LIN {X 0,Y 412.108,Z 841.021,A -85,B 0,C 180,E1 19370.746,E2 19370.746} C_VEL
LIN {X 0,Y 410.858,Z 854.484,A -85,B 0,C 180,E1 19368.885,E2 19368.885} C_VEL
LIN {X 0,Y 409.864,Z 866.557,A -85,B 0,C 180,E1 19366.876,E2 19366.876} C_VEL
LIN {X 0,Y 409.078,Z 878.045,A -85,B 0,C 180,E1 19364.559,E2 19364.559} C_VEL
LIN {X 0,Y 408.646,Z 887.648,A -85,B 0,C 180,E1 19362.147,E2 19362.147} C_VEL
LIN {X 0,Y 408.473,Z 895.28,A -85,B 0,C 180,E1 19359.724,E2 19359.724} C_VEL
LIN {X 0,Y 408.505,Z 901.076,A -85,B 0,C 180,E1 19357.312,E2 19357.312} C_VEL
LIN {X 0,Y 408.633,Z 905.166,A -85,B 0,C 180,E1 19354.913,E2 19354.913} C_VEL
LIN {X 0,Y 408.749,Z 907.618,A -85,B 0,C 180,E1 19352.524,E2 19352.524} C_VEL
LIN {X 0,Y 408.815,Z 908.485,A -85,B 0,C 180,E1 19350,E2 19350} C_VEL
LIN {X 0,Y 408.753,Z 907.591,A -85,B 0,C 180,E1 19347.477,E2 19347.477} C_VEL
LIN {X 0,Y 408.634,Z 904.94,A -85,B 0,C 180,E1 19344.947,E2 19344.947} C_VEL
LIN {X 0,Y 408.493,Z 900.479,A -85,B 0,C 180,E1 19342.405,E2 19342.405} C_VEL
LIN {X 0,Y 408.487,Z 894.1,A -85,B 0,C 180,E1 19339.85,E2 19339.85} C_VEL
LIN {X 0,Y 408.69,Z 886.166,A -85,B 0,C 180,E1 19337.424,E2 19337.424} C_VEL
LIN {X 0,Y 409.156,Z 876.808,A -85,B 0,C 180,E1 19335.132,E2 19335.132} C_VEL
LIN {X 0,Y 409.932,Z 866.006,A -85,B 0,C 180,E1 19332.964,E2 19332.964} C_VEL
LIN {X 0,Y 411.042,Z 853.158,A -85,B 0,C 180,E1 19330.829,E2 19330.829} C_VEL
LIN {X 0,Y 412.424,Z 839.094,A -85,B 0,C 180,E1 19328.899,E2 19328.899} C_VEL
LIN {X 0,Y 414.001,Z 823.32,A -85,B 0,C 180,E1 19327.118,E2 19327.118} C_VEL
LIN {X 0,Y 415.652,Z 807.137,A -85,B 0,C 180,E1 19325.635,E2 19325.635} C_VEL
LIN {X 0,Y 417.149,Z 790.974,A -85,B 0,C 180,E1 19324.441,E2 19324.441} C_VEL
LIN {X 0,Y 418.634,Z 773.451,A -85,B 0,C 180,E1 19323.428,E2 19323.428} C_VEL
LIN {X 0,Y 419.933,Z 754.838,A -85,B 0,C 180,E1 19322.636,E2 19322.636} C_VEL
LIN {X 0,Y 420.832,Z 735.86,A -85,B 0,C 180,E1 19322.104,E2 19322.104} C_VEL
LIN {X 0,Y 423.722,Z 562.823,A -85,B 0,C 180,E1 19319.088,E2 19319.088} C_VEL
LIN {X 0,Y 421.288,Z 541.067,A -85,B 0,C 180,E1 19318.453,E2 19318.453} C_VEL
LIN {X 0,Y 426.206,Z 498.135,A -85,B 0,C 180,E1 19314.092,E2 19314.092} C_VEL
LIN {X 0,Y 423.296,Z 488.09,A -85,B 0,C 180,E1 19312.623,E2 19312.623} C_VEL
LIN {X 0,Y 417.623,Z 472.168,A -85,B 0,C 180,E1 19310.008,E2 19310.008} C_VEL
LIN {X 0,Y 412.165,Z 458.735,A -85,B 0,C 180,E1 19307.516,E2 19307.516} C_VEL
LIN {X 0,Y 409.464,Z 451.977,A -85,B 0,C 180,E1 19306.115,E2 19306.115} C_VEL
LIN {X 0,Y 409.438,Z 451.787,A -85,B 0,C 180,E1 19302.187,E2 19302.187} C_VEL
LIN {X 0,Y 409.436,Z 451.789,A -85,B 0,C 180,E1 19298.336,E2 19298.336} C_VEL
LIN {X 0,Y 409.437,Z 451.796,A -85,B 0,C 180,E1 19294.34,E2 19294.34} C_VEL
LIN {X 0,Y 409.439,Z 451.796,A -85,B 0,C 180,E1 19290.364,E2 19290.364} C_VEL
LIN {X 0,Y 409.438,Z 451.794,A -85,B 0,C 180,E1 19286.544,E2 19286.544} C_VEL
LIN {X 0,Y 409.442,Z 451.791,A -85,B 0,C 180,E1 19282.544,E2 19282.544} C_VEL
LIN {X 0,Y 409.433,Z 451.782,A -85,B 0,C 180,E1 19278.646,E2 19278.646} C_VEL
LIN {X 0,Y 409.428,Z 451.775,A -85,B 0,C 180,E1 19274.713,E2 19274.713} C_VEL
LIN {X 0,Y 409.428,Z 451.787,A -85,B 0,C 180,E1 19270.838,E2 19270.838} C_VEL
LIN {X 0,Y 409.427,Z 451.797,A -85,B 0,C 180,E1 19266.872,E2 19266.872} C_VEL
LIN {X 0,Y 409.431,Z 451.793,A -85,B 0,C 180,E1 19262.939,E2 19262.939} C_VEL
LIN {X 0,Y 409.436,Z 451.78,A -85,B 0,C 180,E1 19259.02,E2 19259.02} C_VEL
LIN {X 0,Y 409.434,Z 451.779,A -85,B 0,C 180,E1 19255.097,E2 19255.097} C_VEL
LIN {X 0,Y 409.438,Z 451.784,A -85,B 0,C 180,E1 19251.291,E2 19251.291} C_VEL
LIN {X 0,Y 409.438,Z 451.789,A -85,B 0,C 180,E1 19247.303,E2 19247.303} C_VEL
LIN {X 0,Y 409.441,Z 451.792,A -85,B 0,C 180,E1 19243.398,E2 19243.398} C_VEL
LIN {X 0,Y 409.441,Z 451.788,A -85,B 0,C 180,E1 19239.411,E2 19239.411} C_VEL
LIN {X 0,Y 409.434,Z 451.786,A -85,B 0,C 180,E1 19235.625,E2 19235.625} C_VEL
LIN {X 0,Y 409.429,Z 451.795,A -85,B 0,C 180,E1 19231.721,E2 19231.721} C_VEL
LIN {X 0,Y 409.479,Z 452.064,A -85,B 0,C 180,E1 19229.358,E2 19229.358} C_VEL
LIN {X 0,Y 414.365,Z 466.013,A -85,B 0,C 180,E1 19226.106,E2 19226.106} C_VEL
LIN {X 0,Y 418.718,Z 480.117,A -85,B 0,C 180,E1 19223.125,E2 19223.125} C_VEL
LIN {X 0,Y 421.8,Z 492.439,A -85,B 0,C 180,E1 19220.734,E2 19220.734} C_VEL
LIN {X 0,Y 418.756,Z 520.346,A -85,B 0,C 180,E1 19216.54,E2 19216.54} C_VEL
LIN {X 0,Y 416.088,Z 548.549,A -85,B 0,C 180,E1 19212.379,E2 19212.379} C_VEL
LIN {X 0,Y 415.681,Z 554.248,A -85,B 0,C 180,E1 19211.576,E2 19211.576} C_VEL
LIN {X 0,Y 417.659,Z 564.451,A -85,B 0,C 180,E1 19211.173,E2 19211.173} C_VEL
LIN {X 0,Y 420.599,Z 581.405,A -85,B 0,C 180,E1 19210.622,E2 19210.622} C_VEL
LIN {X 0,Y 418.499,Z 678.205,A -85,B 0,C 180,E1 19208.79,E2 19208.79} C_VEL
LIN {X 0,Y 417.949,Z 694.436,A -85,B 0,C 180,E1 19208.216,E2 19208.216} C_VEL
LIN {X 0,Y 417.211,Z 708.122,A -85,B 0,C 180,E1 19207.497,E2 19207.497} C_VEL
LIN {X 0,Y 416.181,Z 722.203,A -85,B 0,C 180,E1 19206.492,E2 19206.492} C_VEL
LIN {X 0,Y 415.036,Z 734.8,A -85,B 0,C 180,E1 19205.322,E2 19205.322} C_VEL
LIN {X 0,Y 413.801,Z 747.225,A -85,B 0,C 180,E1 19203.845,E2 19203.845} C_VEL
LIN {X 0,Y 412.619,Z 757.902,A -85,B 0,C 180,E1 19202.215,E2 19202.215} C_VEL
LIN {X 0,Y 411.608,Z 766.741,A -85,B 0,C 180,E1 19200.51,E2 19200.51} C_VEL
LIN {X 0,Y 410.668,Z 774.752,A -85,B 0,C 180,E1 19198.485,E2 19198.485} C_VEL
LIN {X 0,Y 409.991,Z 780.564,A -85,B 0,C 180,E1 19196.489,E2 19196.489} C_VEL
LIN {X 0,Y 409.526,Z 784.81,A -85,B 0,C 180,E1 19194.369,E2 19194.369} C_VEL
LIN {X 0,Y 409.251,Z 787.256,A -85,B 0,C 180,E1 19192.187,E2 19192.187} C_VEL
LIN {X 0,Y 409.145,Z 787.957,A -85,B 0,C 180,E1 19190.006,E2 19190.006} C_VEL
LIN {X 0,Y 409.137,Z 787.808,A -85,B 0,C 180,E1 19189.341,E2 19189.341} C_VEL
LIN {X 0,Y 408.18,Z 787.446,A -85,B 0,C 180,E1 19188.262,E2 19188.262} C_VEL
LIN {X 0,Y 404.232,Z 786.122,A -85,B 0,C 180,E1 19186.459,E2 19186.459} C_VEL
LIN {X 0,Y 401.873,Z 784.219,A -85,B 0,C 180,E1 19185.094,E2 19185.094} C_VEL
LIN {X 0,Y 401.627,Z 783.02,A -85,B 0,C 180,E1 19184.483,E2 19184.483} C_VEL
LIN {X 0,Y 402.092,Z 777.918,A -85,B 0,C 180,E1 19182.494,E2 19182.494} C_VEL
LIN {X 0,Y 402.798,Z 770.631,A -85,B 0,C 180,E1 19180.44,E2 19180.44} C_VEL
LIN {X 0,Y 403.609,Z 762.582,A -85,B 0,C 180,E1 19178.691,E2 19178.691} C_VEL
LIN {X 0,Y 404.628,Z 752.359,A -85,B 0,C 180,E1 19176.954,E2 19176.954} C_VEL
LIN {X 0,Y 405.691,Z 741.112,A -85,B 0,C 180,E1 19175.444,E2 19175.444} C_VEL
LIN {X 0,Y 406.794,Z 728.273,A -85,B 0,C 180,E1 19174.087,E2 19174.087} C_VEL
LIN {X 0,Y 407.821,Z 714.219,A -85,B 0,C 180,E1 19172.951,E2 19172.951} C_VEL
LIN {X 0,Y 408.63,Z 700.315,A -85,B 0,C 180,E1 19172.103,E2 19172.103} C_VEL
LIN {X 0,Y 409.274,Z 683.774,A -85,B 0,C 180,E1 19171.408,E2 19171.408} C_VEL
LIN {X 0,Y 409.627,Z 665.81,A -85,B 0,C 180,E1 19170.979,E2 19170.979} C_VEL
LIN {X 0,Y 411.05,Z 579.361,A -85,B 0,C 180,E1 19169.384,E2 19169.384} C_VEL
LIN {X 0,Y 406.705,Z 554.518,A -85,B 0,C 180,E1 19168.626,E2 19168.626} C_VEL
LIN {X 0,Y 408.776,Z 527.92,A -85,B 0,C 180,E1 19164.807,E2 19164.807} C_VEL
LIN {X 0,Y 411.265,Z 500.481,A -85,B 0,C 180,E1 19160.766,E2 19160.766} C_VEL
LIN {X 0,Y 412.101,Z 490.248,A -85,B 0,C 180,E1 19159.232,E2 19159.232} C_VEL
LIN {X 0,Y 407.297,Z 472.284,A -85,B 0,C 180,E1 19155.934,E2 19155.934} C_VEL
LIN {X 0,Y 402.224,Z 455.434,A -85,B 0,C 180,E1 19152.644,E2 19152.644} C_VEL
LIN {X 0,Y 401.461,Z 452.888,A -85,B 0,C 180,E1 19152.063,E2 19152.063} C_VEL
LIN {X 0,Y 401.432,Z 452.768,A -85,B 0,C 180,E1 19148.215,E2 19148.215} C_VEL
LIN {X 0,Y 401.43,Z 452.789,A -85,B 0,C 180,E1 19144.317,E2 19144.317} C_VEL
LIN {X 0,Y 401.426,Z 452.793,A -85,B 0,C 180,E1 19140.376,E2 19140.376} C_VEL
LIN {X 0,Y 401.426,Z 452.791,A -85,B 0,C 180,E1 19136.43,E2 19136.43} C_VEL
LIN {X 0,Y 401.437,Z 452.779,A -85,B 0,C 180,E1 19132.574,E2 19132.574} C_VEL
LIN {X 0,Y 401.467,Z 452.776,A -85,B 0,C 180,E1 19128.89,E2 19128.89} C_VEL
LIN {X 0,Y 401.477,Z 452.791,A -85,B 0,C 180,E1 19124.985,E2 19124.985} C_VEL
LIN {X 0,Y 401.488,Z 452.764,A -85,B 0,C 180,E1 19120.918,E2 19120.918} C_VEL
LIN {X 0,Y 401.487,Z 452.782,A -85,B 0,C 180,E1 19116.925,E2 19116.925} C_VEL
LIN {X 0,Y 401.485,Z 452.766,A -85,B 0,C 180,E1 19112.882,E2 19112.882} C_VEL
LIN {X 0,Y 401.478,Z 452.783,A -85,B 0,C 180,E1 19109.055,E2 19109.055} C_VEL
LIN {X 0,Y 401.461,Z 452.761,A -85,B 0,C 180,E1 19105.207,E2 19105.207} C_VEL
LIN {X 0,Y 401.452,Z 452.789,A -85,B 0,C 180,E1 19101.477,E2 19101.477} C_VEL
LIN {X 0,Y 401.449,Z 452.752,A -85,B 0,C 180,E1 19097.54,E2 19097.54} C_VEL
LIN {X 0,Y 401.456,Z 452.787,A -85,B 0,C 180,E1 19093.54,E2 19093.54} C_VEL
LIN {X 0,Y 401.458,Z 452.761,A -85,B 0,C 180,E1 19089.606,E2 19089.606} C_VEL
LIN {X 0,Y 401.469,Z 452.782,A -85,B 0,C 180,E1 19085.718,E2 19085.718} C_VEL
LIN {X 0,Y 401.48,Z 452.768,A -85,B 0,C 180,E1 19081.856,E2 19081.856} C_VEL
LIN {X 0,Y 401.496,Z 452.774,A -85,B 0,C 180,E1 19078.002,E2 19078.002} C_VEL
LIN {X 0,Y 401.502,Z 452.771,A -85,B 0,C 180,E1 19073.997,E2 19073.997} C_VEL
LIN {X 0,Y 401.502,Z 452.774,A -85,B 0,C 180,E1 19070.106,E2 19070.106} C_VEL
LIN {X 0,Y 401.502,Z 452.768,A -85,B 0,C 180,E1 19066.169,E2 19066.169} C_VEL
LIN {X 0,Y 401.5,Z 452.785,A -85,B 0,C 180,E1 19062.163,E2 19062.163} C_VEL
LIN {X 0,Y 401.497,Z 452.766,A -85,B 0,C 180,E1 19058.219,E2 19058.219} C_VEL
LIN {X 0,Y 401.488,Z 452.779,A -85,B 0,C 180,E1 19054.321,E2 19054.321} C_VEL
LIN {X 0,Y 401.488,Z 452.789,A -85,B 0,C 180,E1 19050.36,E2 19050.36} C_VEL
LIN {X 0,Y 401.485,Z 452.785,A -85,B 0,C 180,E1 19046.436,E2 19046.436} C_VEL
LIN {X 0,Y 401.484,Z 452.786,A -85,B 0,C 180,E1 19042.58,E2 19042.58} C_VEL
LIN {X 0,Y 401.489,Z 452.787,A -85,B 0,C 180,E1 19038.556,E2 19038.556} C_VEL
LIN {X 0,Y 401.49,Z 452.779,A -85,B 0,C 180,E1 19034.582,E2 19034.582} C_VEL
LIN {X 0,Y 401.526,Z 453.016,A -85,B 0,C 180,E1 19032.727,E2 19032.727} C_VEL
LIN {X 0,Y 408.421,Z 472.022,A -85,B 0,C 180,E1 19029.664,E2 19029.664} C_VEL
LIN {X 0,Y 415.923,Z 494.073,A -85,B 0,C 180,E1 19026.463,E2 19026.463} C_VEL
LIN {X 0,Y 417.225,Z 498.2,A -85,B 0,C 180,E1 19025.904,E2 19025.904} C_VEL
LIN {X 0,Y 412.81,Z 540.992,A -85,B 0,C 180,E1 19021.622,E2 19021.622} C_VEL
LIN {X 0,Y 415.431,Z 566.716,A -85,B 0,C 180,E1 19020.959,E2 19020.959} C_VEL
LIN {X 0,Y 412.493,Z 738.8,A -85,B 0,C 180,E1 19017.967,E2 19017.967} C_VEL
LIN {X 0,Y 411.552,Z 757.391,A -85,B 0,C 180,E1 19017.403,E2 19017.403} C_VEL
LIN {X 0,Y 410.372,Z 774.696,A -85,B 0,C 180,E1 19016.636,E2 19016.636} C_VEL
LIN {X 0,Y 408.983,Z 791.545,A -85,B 0,C 180,E1 19015.641,E2 19015.641} C_VEL
LIN {X 0,Y 407.427,Z 808.616,A -85,B 0,C 180,E1 19014.349,E2 19014.349} C_VEL
LIN {X 0,Y 405.858,Z 824.312,A -85,B 0,C 180,E1 19012.872,E2 19012.872} C_VEL
LIN {X 0,Y 404.35,Z 839.602,A -85,B 0,C 180,E1 19011.11,E2 19011.11} C_VEL
LIN {X 0,Y 403.013,Z 853.315,A -85,B 0,C 180,E1 19009.192,E2 19009.192} C_VEL
LIN {X 0,Y 401.932,Z 865.851,A -85,B 0,C 180,E1 19007.07,E2 19007.07} C_VEL
LIN {X 0,Y 401.161,Z 876.529,A -85,B 0,C 180,E1 19004.876,E2 19004.876} C_VEL
LIN {X 0,Y 400.687,Z 886.318,A -85,B 0,C 180,E1 19002.392,E2 19002.392} C_VEL
LIN {X 0,Y 400.51,Z 894.001,A -85,B 0,C 180,E1 18999.919,E2 18999.919} C_VEL
LIN {X 0,Y 400.548,Z 899.837,A -85,B 0,C 180,E1 18997.459,E2 18997.459} C_VEL
LIN {X 0,Y 400.697,Z 903.962,A -85,B 0,C 180,E1 18995.011,E2 18995.011} C_VEL
LIN {X 0,Y 400.836,Z 906.525,A -85,B 0,C 180,E1 18992.431,E2 18992.431} C_VEL
LIN {X 0,Y 400.897,Z 907.312,A -85,B 0,C 180,E1 18989.857,E2 18989.857} C_VEL
LIN {X 0,Y 400.823,Z 906.329,A -85,B 0,C 180,E1 18987.284,E2 18987.284} C_VEL
LIN {X 0,Y 400.676,Z 903.574,A -85,B 0,C 180,E1 18984.703,E2 18984.703} C_VEL
LIN {X 0,Y 400.524,Z 898.987,A -85,B 0,C 180,E1 18982.109,E2 18982.109} C_VEL
LIN {X 0,Y 400.516,Z 892.781,A -85,B 0,C 180,E1 18979.606,E2 18979.606} C_VEL
LIN {X 0,Y 400.732,Z 884.94,A -85,B 0,C 180,E1 18977.17,E2 18977.17} C_VEL
LIN {X 0,Y 401.238,Z 875.583,A -85,B 0,C 180,E1 18974.832,E2 18974.832} C_VEL
LIN {X 0,Y 402.063,Z 864.886,A -85,B 0,C 180,E1 18972.638,E2 18972.638} C_VEL
LIN {X 0,Y 403.172,Z 852.878,A -85,B 0,C 180,E1 18970.591,E2 18970.591} C_VEL
LIN {X 0,Y 404.624,Z 838.96,A -85,B 0,C 180,E1 18968.624,E2 18968.624} C_VEL
LIN {X 0,Y 406.209,Z 824.047,A -85,B 0,C 180,E1 18966.884,E2 18966.884} C_VEL
LIN {X 0,Y 408.013,Z 807.384,A -85,B 0,C 180,E1 18965.303,E2 18965.303} C_VEL
LIN {X 0,Y 409.667,Z 790.598,A -85,B 0,C 180,E1 18964.028,E2 18964.028} C_VEL
LIN {X 0,Y 411.178,Z 773.845,A -85,B 0,C 180,E1 18963.031,E2 18963.031} C_VEL
LIN {X 0,Y 412.528,Z 755.816,A -85,B 0,C 180,E1 18962.229,E2 18962.229} C_VEL
LIN {X 0,Y 413.534,Z 737.11,A -85,B 0,C 180,E1 18961.667,E2 18961.667} C_VEL
LIN {X 0,Y 416.67,Z 563.768,A -85,B 0,C 180,E1 18958.584,E2 18958.584} C_VEL
LIN {X 0,Y 414.152,Z 541.339,A -85,B 0,C 180,E1 18957.918,E2 18957.918} C_VEL
LIN {X 0,Y 419.123,Z 500.336,A -85,B 0,C 180,E1 18953.662,E2 18953.662} C_VEL
LIN {X 0,Y 413.776,Z 483.941,A -85,B 0,C 180,E1 18951.078,E2 18951.078} C_VEL
LIN {X 0,Y 407.629,Z 467.636,A -85,B 0,C 180,E1 18948.151,E2 18948.151} C_VEL
LIN {X 0,Y 402.535,Z 455.853,A -85,B 0,C 180,E1 18945.735,E2 18945.735} C_VEL
LIN {X 0,Y 401.519,Z 452.934,A -85,B 0,C 180,E1 18945.053,E2 18945.053} C_VEL
LIN {X 0,Y 401.506,Z 452.783,A -85,B 0,C 180,E1 18941.014,E2 18941.014} C_VEL
LIN {X 0,Y 401.496,Z 452.785,A -85,B 0,C 180,E1 18937.06,E2 18937.06} C_VEL
LIN {X 0,Y 401.494,Z 452.777,A -85,B 0,C 180,E1 18933.051,E2 18933.051} C_VEL
LIN {X 0,Y 401.493,Z 452.775,A -85,B 0,C 180,E1 18929.053,E2 18929.053} C_VEL
LIN {X 0,Y 401.491,Z 452.778,A -85,B 0,C 180,E1 18925.047,E2 18925.047} C_VEL
LIN {X 0,Y 401.491,Z 452.782,A -85,B 0,C 180,E1 18921.015,E2 18921.015} C_VEL
LIN {X 0,Y 401.49,Z 452.787,A -85,B 0,C 180,E1 18917.001,E2 18917.001} C_VEL
LIN {X 0,Y 401.492,Z 452.777,A -85,B 0,C 180,E1 18913.098,E2 18913.098} C_VEL
LIN {X 0,Y 401.493,Z 452.767,A -85,B 0,C 180,E1 18909.171,E2 18909.171} C_VEL
LIN {X 0,Y 401.496,Z 452.767,A -85,B 0,C 180,E1 18905.287,E2 18905.287} C_VEL
LIN {X 0,Y 401.502,Z 452.779,A -85,B 0,C 180,E1 18901.284,E2 18901.284} C_VEL
LIN {X 0,Y 401.499,Z 452.787,A -85,B 0,C 180,E1 18897.288,E2 18897.288} C_VEL
LIN {X 0,Y 401.503,Z 452.78,A -85,B 0,C 180,E1 18893.278,E2 18893.278} C_VEL
LIN {X 0,Y 401.499,Z 452.776,A -85,B 0,C 180,E1 18889.235,E2 18889.235} C_VEL
LIN {X 0,Y 401.502,Z 452.774,A -85,B 0,C 180,E1 18885.285,E2 18885.285} C_VEL
LIN {X 0,Y 401.501,Z 452.778,A -85,B 0,C 180,E1 18881.261,E2 18881.261} C_VEL
LIN {X 0,Y 401.506,Z 452.785,A -85,B 0,C 180,E1 18877.294,E2 18877.294} C_VEL
LIN {X 0,Y 401.5,Z 452.78,A -85,B 0,C 180,E1 18873.368,E2 18873.368} C_VEL
LIN {X 0,Y 401.536,Z 453.052,A -85,B 0,C 180,E1 18870.359,E2 18870.359} C_VEL
LIN {X 0,Y 406.172,Z 465.882,A -85,B 0,C 180,E1 18867.209,E2 18867.209} C_VEL
LIN {X 0,Y 410.698,Z 480.056,A -85,B 0,C 180,E1 18864.075,E2 18864.075} C_VEL
LIN {X 0,Y 414.48,Z 494.529,A -85,B 0,C 180,E1 18861.155,E2 18861.155} C_VEL
LIN {X 0,Y 412.074,Z 516.12,A -85,B 0,C 180,E1 18857.839,E2 18857.839} C_VEL
LIN {X 0,Y 409.252,Z 543.685,A -85,B 0,C 180,E1 18853.683,E2 18853.683} C_VEL
LIN {X 0,Y 408.353,Z 554.376,A -85,B 0,C 180,E1 18852.136,E2 18852.136} C_VEL
LIN {X 0,Y 413.566,Z 581.773,A -85,B 0,C 180,E1 18851.143,E2 18851.143} C_VEL
LIN {X 0,Y 411.336,Z 678.782,A -85,B 0,C 180,E1 18849.276,E2 18849.276} C_VEL
LIN {X 0,Y 410.757,Z 694.919,A -85,B 0,C 180,E1 18848.698,E2 18848.698} C_VEL
LIN {X 0,Y 409.931,Z 709.332,A -85,B 0,C 180,E1 18847.926,E2 18847.926} C_VEL
LIN {X 0,Y 408.832,Z 723.463,A -85,B 0,C 180,E1 18846.895,E2 18846.895} C_VEL
LIN {X 0,Y 407.627,Z 735.875,A -85,B 0,C 180,E1 18845.717,E2 18845.717} C_VEL
LIN {X 0,Y 406.313,Z 748.189,A -85,B 0,C 180,E1 18844.224,E2 18844.224} C_VEL
LIN {X 0,Y 405.035,Z 758.912,A -85,B 0,C 180,E1 18842.557,E2 18842.557} C_VEL
LIN {X 0,Y 403.933,Z 767.836,A -85,B 0,C 180,E1 18840.802,E2 18840.802} C_VEL
LIN {X 0,Y 402.929,Z 775.709,A -85,B 0,C 180,E1 18838.777,E2 18838.777} C_VEL
LIN {X 0,Y 402.189,Z 781.578,A -85,B 0,C 180,E1 18836.742,E2 18836.742} C_VEL
LIN {X 0,Y 401.667,Z 785.892,A -85,B 0,C 180,E1 18834.564,E2 18834.564} C_VEL
LIN {X 0,Y 401.366,Z 788.34,A -85,B 0,C 180,E1 18832.404,E2 18832.404} C_VEL
LIN {X 0,Y 401.234,Z 789.138,A -85,B 0,C 180,E1 18830.114,E2 18830.114} C_VEL
LIN {X 0,Y 401.257,Z 788.058,A -85,B 0,C 180,E1 18827.846,E2 18827.846} C_VEL
LIN {X 0,Y 401.44,Z 785.457,A -85,B 0,C 180,E1 18825.752,E2 18825.752} C_VEL
LIN {X 0,Y 401.627,Z 783.02,A -85,B 0,C 180,E1 18824.483,E2 18824.483} C_VEL
LIN {X 0,Y 400.869,Z 780.731,A -85,B 0,C 180,E1 18823.427,E2 18823.427} C_VEL
LIN {X 0,Y 397.327,Z 776.403,A -85,B 0,C 180,E1 18821.672,E2 18821.672} C_VEL
LIN {X 0,Y 395.285,Z 772.231,A -85,B 0,C 180,E1 18820.385,E2 18820.385} C_VEL
LIN {X 0,Y 395.166,Z 769.988,A -85,B 0,C 180,E1 18819.829,E2 18819.829} C_VEL
LIN {X 0,Y 396.107,Z 761.081,A -85,B 0,C 180,E1 18817.98,E2 18817.98} C_VEL
LIN {X 0,Y 397.189,Z 750.691,A -85,B 0,C 180,E1 18816.286,E2 18816.286} C_VEL
LIN {X 0,Y 398.347,Z 738.786,A -85,B 0,C 180,E1 18814.751,E2 18814.751} C_VEL
LIN {X 0,Y 399.478,Z 725.741,A -85,B 0,C 180,E1 18813.444,E2 18813.444} C_VEL
LIN {X 0,Y 400.504,Z 711.738,A -85,B 0,C 180,E1 18812.361,E2 18812.361} C_VEL
LIN {X 0,Y 401.349,Z 696.534,A -85,B 0,C 180,E1 18811.499,E2 18811.499} C_VEL
LIN {X 0,Y 401.896,Z 681.019,A -85,B 0,C 180,E1 18810.909,E2 18810.909} C_VEL
LIN {X 0,Y 402.432,Z 653.413,A -85,B 0,C 180,E1 18810.324,E2 18810.324} C_VEL
LIN {X 0,Y 403.659,Z 580.369,A -85,B 0,C 180,E1 18808.957,E2 18808.957} C_VEL
LIN {X 0,Y 399.141,Z 554.231,A -85,B 0,C 180,E1 18808.134,E2 18808.134} C_VEL
LIN {X 0,Y 401.425,Z 526.958,A -85,B 0,C 180,E1 18804.138,E2 18804.138} C_VEL
LIN {X 0,Y 404.097,Z 499.455,A -85,B 0,C 180,E1 18800.026,E2 18800.026} C_VEL
LIN {X 0,Y 404.665,Z 492.91,A -85,B 0,C 180,E1 18799.032,E2 18799.032} C_VEL
LIN {X 0,Y 400.117,Z 475.734,A -85,B 0,C 180,E1 18795.824,E2 18795.824} C_VEL
LIN {X 0,Y 395.046,Z 458.853,A -85,B 0,C 180,E1 18792.471,E2 18792.471} C_VEL
LIN {X 0,Y 393.548,Z 453.877,A -85,B 0,C 180,E1 18791.381,E2 18791.381} C_VEL
LIN {X 0,Y 393.544,Z 453.735,A -85,B 0,C 180,E1 18787.44,E2 18787.44} C_VEL
LIN {X 0,Y 393.536,Z 453.78,A -85,B 0,C 180,E1 18783.423,E2 18783.423} C_VEL
LIN {X 0,Y 393.533,Z 453.779,A -85,B 0,C 180,E1 18779.459,E2 18779.459} C_VEL
LIN {X 0,Y 393.527,Z 453.781,A -85,B 0,C 180,E1 18775.408,E2 18775.408} C_VEL
LIN {X 0,Y 393.535,Z 453.774,A -85,B 0,C 180,E1 18771.316,E2 18771.316} C_VEL
LIN {X 0,Y 393.516,Z 453.758,A -85,B 0,C 180,E1 18767.464,E2 18767.464} C_VEL
LIN {X 0,Y 393.508,Z 453.779,A -85,B 0,C 180,E1 18763.601,E2 18763.601} C_VEL
LIN {X 0,Y 393.501,Z 453.77,A -85,B 0,C 180,E1 18759.816,E2 18759.816} C_VEL
LIN {X 0,Y 393.501,Z 453.769,A -85,B 0,C 180,E1 18755.849,E2 18755.849} C_VEL
LIN {X 0,Y 393.506,Z 453.773,A -85,B 0,C 180,E1 18751.905,E2 18751.905} C_VEL
LIN {X 0,Y 393.512,Z 453.765,A -85,B 0,C 180,E1 18748.039,E2 18748.039} C_VEL
LIN {X 0,Y 393.522,Z 453.767,A -85,B 0,C 180,E1 18744.147,E2 18744.147} C_VEL
LIN {X 0,Y 393.546,Z 453.766,A -85,B 0,C 180,E1 18740.364,E2 18740.364} C_VEL
LIN {X 0,Y 393.551,Z 453.746,A -85,B 0,C 180,E1 18736.38,E2 18736.38} C_VEL
LIN {X 0,Y 393.558,Z 453.772,A -85,B 0,C 180,E1 18732.471,E2 18732.471} C_VEL
LIN {X 0,Y 393.557,Z 453.738,A -85,B 0,C 180,E1 18728.474,E2 18728.474} C_VEL
LIN {X 0,Y 393.555,Z 453.776,A -85,B 0,C 180,E1 18724.517,E2 18724.517} C_VEL
LIN {X 0,Y 393.559,Z 453.74,A -85,B 0,C 180,E1 18720.437,E2 18720.437} C_VEL
LIN {X 0,Y 393.55,Z 453.775,A -85,B 0,C 180,E1 18716.505,E2 18716.505} C_VEL
LIN {X 0,Y 393.543,Z 453.748,A -85,B 0,C 180,E1 18712.555,E2 18712.555} C_VEL
LIN {X 0,Y 393.543,Z 453.776,A -85,B 0,C 180,E1 18708.57,E2 18708.57} C_VEL
LIN {X 0,Y 393.536,Z 453.751,A -85,B 0,C 180,E1 18704.679,E2 18704.679} C_VEL
LIN {X 0,Y 393.54,Z 453.777,A -85,B 0,C 180,E1 18700.714,E2 18700.714} C_VEL
LIN {X 0,Y 393.539,Z 453.769,A -85,B 0,C 180,E1 18696.809,E2 18696.809} C_VEL
LIN {X 0,Y 393.538,Z 453.757,A -85,B 0,C 180,E1 18692.779,E2 18692.779} C_VEL
LIN {X 0,Y 393.544,Z 453.764,A -85,B 0,C 180,E1 18688.782,E2 18688.782} C_VEL
LIN {X 0,Y 393.545,Z 453.767,A -85,B 0,C 180,E1 18684.78,E2 18684.78} C_VEL
LIN {X 0,Y 393.548,Z 453.765,A -85,B 0,C 180,E1 18680.757,E2 18680.757} C_VEL
LIN {X 0,Y 393.555,Z 453.769,A -85,B 0,C 180,E1 18676.815,E2 18676.815} C_VEL
LIN {X 0,Y 393.597,Z 454.026,A -85,B 0,C 180,E1 18673.457,E2 18673.457} C_VEL
LIN {X 0,Y 400.542,Z 473.077,A -85,B 0,C 180,E1 18670.281,E2 18670.281} C_VEL
LIN {X 0,Y 407.843,Z 494.443,A -85,B 0,C 180,E1 18667.092,E2 18667.092} C_VEL
LIN {X 0,Y 409.804,Z 500.937,A -85,B 0,C 180,E1 18666.189,E2 18666.189} C_VEL
LIN {X 0,Y 405.429,Z 541.304,A -85,B 0,C 180,E1 18662.077,E2 18662.077} C_VEL
LIN {X 0,Y 408.091,Z 567.582,A -85,B 0,C 180,E1 18661.393,E2 18661.393} C_VEL
LIN {X 0,Y 405.048,Z 738.109,A -85,B 0,C 180,E1 18658.387,E2 18658.387} C_VEL
LIN {X 0,Y 404.074,Z 756.704,A -85,B 0,C 180,E1 18657.813,E2 18657.813} C_VEL
LIN {X 0,Y 402.817,Z 774.328,A -85,B 0,C 180,E1 18657.016,E2 18657.016} C_VEL
LIN {X 0,Y 401.261,Z 792.231,A -85,B 0,C 180,E1 18655.925,E2 18655.925} C_VEL
LIN {X 0,Y 399.659,Z 808.92,A -85,B 0,C 180,E1 18654.617,E2 18654.617} C_VEL
LIN {X 0,Y 397.995,Z 824.776,A -85,B 0,C 180,E1 18653.074,E2 18653.074} C_VEL
LIN {X 0,Y 396.453,Z 839.691,A -85,B 0,C 180,E1 18651.295,E2 18651.295} C_VEL
LIN {X 0,Y 395.087,Z 853.081,A -85,B 0,C 180,E1 18649.362,E2 18649.362} C_VEL
LIN {X 0,Y 393.94,Z 865.854,A -85,B 0,C 180,E1 18647.123,E2 18647.123} C_VEL
LIN {X 0,Y 393.162,Z 876.344,A -85,B 0,C 180,E1 18644.884,E2 18644.884} C_VEL
LIN {X 0,Y 392.713,Z 885.455,A -85,B 0,C 180,E1 18642.499,E2 18642.499} C_VEL
LIN {X 0,Y 392.544,Z 893.096,A -85,B 0,C 180,E1 18639.974,E2 18639.974} C_VEL
LIN {X 0,Y 392.598,Z 898.872,A -85,B 0,C 180,E1 18637.463,E2 18637.463} C_VEL
LIN {X 0,Y 392.77,Z 902.929,A -85,B 0,C 180,E1 18634.966,E2 18634.966} C_VEL
LIN {X 0,Y 392.914,Z 905.343,A -85,B 0,C 180,E1 18632.48,E2 18632.48} C_VEL
LIN {X 0,Y 392.988,Z 906.14,A -85,B 0,C 180,E1 18630,E2 18630} C_VEL
LIN {X 0,Y 392.915,Z 905.337,A -85,B 0,C 180,E1 18627.521,E2 18627.521} C_VEL
LIN {X 0,Y 392.768,Z 902.957,A -85,B 0,C 180,E1 18625.035,E2 18625.035} C_VEL
LIN {X 0,Y 392.589,Z 898.957,A -85,B 0,C 180,E1 18622.537,E2 18622.537} C_VEL
LIN {X 0,Y 392.528,Z 893.275,A -85,B 0,C 180,E1 18620.026,E2 18620.026} C_VEL
LIN {X 0,Y 392.695,Z 885.785,A -85,B 0,C 180,E1 18617.501,E2 18617.501} C_VEL
LIN {X 0,Y 393.191,Z 876.288,A -85,B 0,C 180,E1 18614.967,E2 18614.967} C_VEL
LIN {X 0,Y 394.092,Z 865.066,A -85,B 0,C 180,E1 18612.546,E2 18612.546} C_VEL
LIN {X 0,Y 395.311,Z 852.598,A -85,B 0,C 180,E1 18610.343,E2 18610.343} C_VEL
LIN {X 0,Y 396.834,Z 838.825,A -85,B 0,C 180,E1 18608.339,E2 18608.339} C_VEL
LIN {X 0,Y 398.501,Z 824.099,A -85,B 0,C 180,E1 18606.567,E2 18606.567} C_VEL
LIN {X 0,Y 400.302,Z 808.551,A -85,B 0,C 180,E1 18605.032,E2 18605.032} C_VEL
LIN {X 0,Y 402.038,Z 792.182,A -85,B 0,C 180,E1 18603.725,E2 18603.725} C_VEL
LIN {X 0,Y 403.705,Z 774.988,A -85,B 0,C 180,E1 18602.65,E2 18602.65} C_VEL
LIN {X 0,Y 405.199,Z 756.378,A -85,B 0,C 180,E1 18601.786,E2 18601.786} C_VEL
LIN {X 0,Y 406.276,Z 737.933,A -85,B 0,C 180,E1 18601.206,E2 18601.206} C_VEL
LIN {X 0,Y 407.13,Z 697.172,A -85,B 0,C 180,E1 18600.456,E2 18600.456} C_VEL
LIN {X 0,Y 409.654,Z 564.686,A -85,B 0,C 180,E1 18598.06,E2 18598.06} C_VEL
LIN {X 0,Y 407.071,Z 541.874,A -85,B 0,C 180,E1 18597.375,E2 18597.375} C_VEL
LIN {X 0,Y 412.013,Z 503.231,A -85,B 0,C 180,E1 18593.296,E2 18593.296} C_VEL
LIN {X 0,Y 406.716,Z 486.818,A -85,B 0,C 180,E1 18590.635,E2 18590.635} C_VEL
LIN {X 0,Y 400.899,Z 471.491,A -85,B 0,C 180,E1 18587.793,E2 18587.793} C_VEL
LIN {X 0,Y 396.029,Z 460.11,A -85,B 0,C 180,E1 18585.395,E2 18585.395} C_VEL
LIN {X 0,Y 393.583,Z 453.942,A -85,B 0,C 180,E1 18583.966,E2 18583.966} C_VEL
LIN {X 0,Y 393.563,Z 453.767,A -85,B 0,C 180,E1 18579.997,E2 18579.997} C_VEL
LIN {X 0,Y 393.557,Z 453.761,A -85,B 0,C 180,E1 18575.935,E2 18575.935} C_VEL
LIN {X 0,Y 393.56,Z 453.759,A -85,B 0,C 180,E1 18571.947,E2 18571.947} C_VEL
LIN {X 0,Y 393.561,Z 453.756,A -85,B 0,C 180,E1 18568.034,E2 18568.034} C_VEL
LIN {X 0,Y 393.56,Z 453.755,A -85,B 0,C 180,E1 18563.984,E2 18563.984} C_VEL
LIN {X 0,Y 393.56,Z 453.757,A -85,B 0,C 180,E1 18559.949,E2 18559.949} C_VEL
LIN {X 0,Y 393.562,Z 453.765,A -85,B 0,C 180,E1 18555.925,E2 18555.925} C_VEL
LIN {X 0,Y 393.561,Z 453.775,A -85,B 0,C 180,E1 18551.875,E2 18551.875} C_VEL
LIN {X 0,Y 393.562,Z 453.769,A -85,B 0,C 180,E1 18547.885,E2 18547.885} C_VEL
LIN {X 0,Y 393.557,Z 453.755,A -85,B 0,C 180,E1 18543.933,E2 18543.933} C_VEL
LIN {X 0,Y 393.567,Z 453.752,A -85,B 0,C 180,E1 18539.854,E2 18539.854} C_VEL
LIN {X 0,Y 393.558,Z 453.76,A -85,B 0,C 180,E1 18535.775,E2 18535.775} C_VEL
LIN {X 0,Y 393.563,Z 453.769,A -85,B 0,C 180,E1 18531.82,E2 18531.82} C_VEL
LIN {X 0,Y 393.557,Z 453.773,A -85,B 0,C 180,E1 18527.826,E2 18527.826} C_VEL
LIN {X 0,Y 393.557,Z 453.774,A -85,B 0,C 180,E1 18523.808,E2 18523.808} C_VEL
LIN {X 0,Y 393.555,Z 453.771,A -85,B 0,C 180,E1 18519.786,E2 18519.786} C_VEL
LIN {X 0,Y 393.549,Z 453.765,A -85,B 0,C 180,E1 18515.855,E2 18515.855} C_VEL
LIN {X 0,Y 393.55,Z 453.77,A -85,B 0,C 180,E1 18511.799,E2 18511.799} C_VEL
LIN {X 0,Y 393.625,Z 454.167,A -85,B 0,C 180,E1 18511.392,E2 18511.392} C_VEL
LIN {X 0,Y 398.248,Z 466.644,A -85,B 0,C 180,E1 18508.181,E2 18508.181} C_VEL
LIN {X 0,Y 402.702,Z 480.398,A -85,B 0,C 180,E1 18505.002,E2 18505.002} C_VEL
LIN {X 0,Y 406.421,Z 493.903,A -85,B 0,C 180,E1 18502.158,E2 18502.158} C_VEL
LIN {X 0,Y 407.275,Z 498.66,A -85,B 0,C 180,E1 18501.242,E2 18501.242} C_VEL
LIN {X 0,Y 403.885,Z 526.615,A -85,B 0,C 180,E1 18496.911,E2 18496.911} C_VEL
LIN {X 0,Y 401.055,Z 553.776,A -85,B 0,C 180,E1 18492.79,E2 18492.79} C_VEL
LIN {X 0,Y 402.215,Z 559.867,A -85,B 0,C 180,E1 18492.504,E2 18492.504} C_VEL
LIN {X 0,Y 406.539,Z 583.602,A -85,B 0,C 180,E1 18491.656,E2 18491.656} C_VEL
LIN {X 0,Y 404.202,Z 679.474,A -85,B 0,C 180,E1 18489.776,E2 18489.776} C_VEL
LIN {X 0,Y 403.587,Z 695.623,A -85,B 0,C 180,E1 18489.187,E2 18489.187} C_VEL
LIN {X 0,Y 402.771,Z 709.323,A -85,B 0,C 180,E1 18488.451,E2 18488.451} C_VEL
LIN {X 0,Y 401.602,Z 723.583,A -85,B 0,C 180,E1 18487.407,E2 18487.407} C_VEL
LIN {X 0,Y 400.343,Z 736.053,A -85,B 0,C 180,E1 18486.225,E2 18486.225} C_VEL
LIN {X 0,Y 398.895,Z 748.715,A -85,B 0,C 180,E1 18484.68,E2 18484.68} C_VEL
LIN {X 0,Y 397.594,Z 759.051,A -85,B 0,C 180,E1 18483.073,E2 18483.073} C_VEL
LIN {X 0,Y 396.301,Z 768.801,A -85,B 0,C 180,E1 18481.145,E2 18481.145} C_VEL
LIN {X 0,Y 395.202,Z 776.773,A -85,B 0,C 180,E1 18479.062,E2 18479.062} C_VEL
LIN {X 0,Y 394.394,Z 782.659,A -85,B 0,C 180,E1 18476.987,E2 18476.987} C_VEL
LIN {X 0,Y 393.791,Z 787.202,A -85,B 0,C 180,E1 18474.634,E2 18474.634} C_VEL
LIN {X 0,Y 393.452,Z 789.638,A -85,B 0,C 180,E1 18472.328,E2 18472.328} C_VEL
LIN {X 0,Y 393.319,Z 790.302,A -85,B 0,C 180,E1 18470.071,E2 18470.071} C_VEL
LIN {X 0,Y 393.357,Z 789.026,A -85,B 0,C 180,E1 18467.597,E2 18467.597} C_VEL
LIN {X 0,Y 393.56,Z 786.226,A -85,B 0,C 180,E1 18465.471,E2 18465.471} C_VEL
LIN {X 0,Y 393.997,Z 781.396,A -85,B 0,C 180,E1 18463.202,E2 18463.202} C_VEL
LIN {X 0,Y 394.643,Z 774.929,A -85,B 0,C 180,E1 18461.102,E2 18461.102} C_VEL
LIN {X 0,Y 395.166,Z 769.988,A -85,B 0,C 180,E1 18459.829,E2 18459.829} C_VEL
LIN {X 0,Y 394.624,Z 765.937,A -85,B 0,C 180,E1 18458.878,E2 18458.878} C_VEL
LIN {X 0,Y 390.948,Z 757.492,A -85,B 0,C 180,E1 18457.034,E2 18457.034} C_VEL
LIN {X 0,Y 389.664,Z 751.849,A -85,B 0,C 180,E1 18456.037,E2 18456.037} C_VEL
LIN {X 0,Y 389.727,Z 749.48,A -85,B 0,C 180,E1 18455.684,E2 18455.684} C_VEL
LIN {X 0,Y 390.917,Z 737.466,A -85,B 0,C 180,E1 18454.18,E2 18454.18} C_VEL
LIN {X 0,Y 392.072,Z 724.729,A -85,B 0,C 180,E1 18452.923,E2 18452.923} C_VEL
LIN {X 0,Y 393.07,Z 711.171,A -85,B 0,C 180,E1 18451.895,E2 18451.895} C_VEL
LIN {X 0,Y 393.937,Z 695.871,A -85,B 0,C 180,E1 18451.036,E2 18451.036} C_VEL
LIN {X 0,Y 394.524,Z 678.973,A -85,B 0,C 180,E1 18450.417,E2 18450.417} C_VEL
LIN {X 0,Y 396.301,Z 581.426,A -85,B 0,C 180,E1 18448.517,E2 18448.517} C_VEL
LIN {X 0,Y 391.627,Z 554.389,A -85,B 0,C 180,E1 18447.659,E2 18447.659} C_VEL
LIN {X 0,Y 391.986,Z 549.093,A -85,B 0,C 180,E1 18446.929,E2 18446.929} C_VEL
LIN {X 0,Y 394.602,Z 521.166,A -85,B 0,C 180,E1 18442.721,E2 18442.721} C_VEL
LIN {X 0,Y 397.227,Z 495.556,A -85,B 0,C 180,E1 18438.824,E2 18438.824} C_VEL
LIN {X 0,Y 392.542,Z 477.82,A -85,B 0,C 180,E1 18435.448,E2 18435.448} C_VEL
LIN {X 0,Y 387.889,Z 462.262,A -85,B 0,C 180,E1 18432.292,E2 18432.292} C_VEL
LIN {X 0,Y 385.572,Z 454.885,A -85,B 0,C 180,E1 18430.665,E2 18430.665} C_VEL
LIN {X 0,Y 385.551,Z 454.725,A -85,B 0,C 180,E1 18426.642,E2 18426.642} C_VEL
LIN {X 0,Y 385.556,Z 454.766,A -85,B 0,C 180,E1 18422.676,E2 18422.676} C_VEL
LIN {X 0,Y 385.56,Z 454.763,A -85,B 0,C 180,E1 18418.758,E2 18418.758} C_VEL
LIN {X 0,Y 385.568,Z 454.765,A -85,B 0,C 180,E1 18414.773,E2 18414.773} C_VEL
LIN {X 0,Y 385.575,Z 454.77,A -85,B 0,C 180,E1 18410.748,E2 18410.748} C_VEL
LIN {X 0,Y 385.581,Z 454.752,A -85,B 0,C 180,E1 18406.775,E2 18406.775} C_VEL
LIN {X 0,Y 385.592,Z 454.75,A -85,B 0,C 180,E1 18402.791,E2 18402.791} C_VEL
LIN {X 0,Y 385.612,Z 454.762,A -85,B 0,C 180,E1 18398.865,E2 18398.865} C_VEL
LIN {X 0,Y 385.6,Z 454.734,A -85,B 0,C 180,E1 18394.783,E2 18394.783} C_VEL
LIN {X 0,Y 385.619,Z 454.766,A -85,B 0,C 180,E1 18390.717,E2 18390.717} C_VEL
LIN {X 0,Y 385.608,Z 454.729,A -85,B 0,C 180,E1 18386.653,E2 18386.653} C_VEL
LIN {X 0,Y 385.625,Z 454.764,A -85,B 0,C 180,E1 18382.566,E2 18382.566} C_VEL
LIN {X 0,Y 385.609,Z 454.728,A -85,B 0,C 180,E1 18378.442,E2 18378.442} C_VEL
LIN {X 0,Y 385.625,Z 454.758,A -85,B 0,C 180,E1 18374.413,E2 18374.413} C_VEL
LIN {X 0,Y 385.615,Z 454.738,A -85,B 0,C 180,E1 18370.307,E2 18370.307} C_VEL
LIN {X 0,Y 385.621,Z 454.75,A -85,B 0,C 180,E1 18366.252,E2 18366.252} C_VEL
LIN {X 0,Y 385.619,Z 454.746,A -85,B 0,C 180,E1 18362.229,E2 18362.229} C_VEL
LIN {X 0,Y 385.623,Z 454.745,A -85,B 0,C 180,E1 18358.217,E2 18358.217} C_VEL
LIN {X 0,Y 385.623,Z 454.751,A -85,B 0,C 180,E1 18354.197,E2 18354.197} C_VEL
LIN {X 0,Y 385.622,Z 454.749,A -85,B 0,C 180,E1 18350.147,E2 18350.147} C_VEL
LIN {X 0,Y 385.628,Z 454.743,A -85,B 0,C 180,E1 18346.047,E2 18346.047} C_VEL
LIN {X 0,Y 385.625,Z 454.764,A -85,B 0,C 180,E1 18342.029,E2 18342.029} C_VEL
LIN {X 0,Y 385.629,Z 454.742,A -85,B 0,C 180,E1 18337.917,E2 18337.917} C_VEL
LIN {X 0,Y 385.623,Z 454.747,A -85,B 0,C 180,E1 18333.846,E2 18333.846} C_VEL
LIN {X 0,Y 385.629,Z 454.759,A -85,B 0,C 180,E1 18329.801,E2 18329.801} C_VEL
LIN {X 0,Y 385.623,Z 454.762,A -85,B 0,C 180,E1 18325.761,E2 18325.761} C_VEL
LIN {X 0,Y 385.625,Z 454.759,A -85,B 0,C 180,E1 18321.707,E2 18321.707} C_VEL
LIN {X 0,Y 385.623,Z 454.754,A -85,B 0,C 180,E1 18317.613,E2 18317.613} C_VEL
LIN {X 0,Y 385.649,Z 455.008,A -85,B 0,C 180,E1 18314.221,E2 18314.221} C_VEL
LIN {X 0,Y 392.594,Z 473.89,A -85,B 0,C 180,E1 18310.964,E2 18310.964} C_VEL
LIN {X 0,Y 399.68,Z 494.605,A -85,B 0,C 180,E1 18307.766,E2 18307.766} C_VEL
LIN {X 0,Y 402.437,Z 503.273,A -85,B 0,C 180,E1 18306.525,E2 18306.525} C_VEL
LIN {X 0,Y 398.069,Z 541.441,A -85,B 0,C 180,E1 18302.558,E2 18302.558} C_VEL
LIN {X 0,Y 400.76,Z 568.435,A -85,B 0,C 180,E1 18301.838,E2 18301.838} C_VEL
LIN {X 0,Y 397.581,Z 737.598,A -85,B 0,C 180,E1 18298.803,E2 18298.803} C_VEL
LIN {X 0,Y 396.581,Z 756.138,A -85,B 0,C 180,E1 18298.222,E2 18298.222} C_VEL
LIN {X 0,Y 395.224,Z 774.342,A -85,B 0,C 180,E1 18297.38,E2 18297.38} C_VEL
LIN {X 0,Y 393.619,Z 792.035,A -85,B 0,C 180,E1 18296.275,E2 18296.275} C_VEL
LIN {X 0,Y 391.989,Z 808.345,A -85,B 0,C 180,E1 18294.97,E2 18294.97} C_VEL
LIN {X 0,Y 390.25,Z 824.168,A -85,B 0,C 180,E1 18293.399,E2 18293.399} C_VEL
LIN {X 0,Y 388.637,Z 839.024,A -85,B 0,C 180,E1 18291.587,E2 18291.587} C_VEL
LIN {X 0,Y 387.211,Z 852.36,A -85,B 0,C 180,E1 18289.615,E2 18289.615} C_VEL
LIN {X 0,Y 386.014,Z 865.06,A -85,B 0,C 180,E1 18287.33,E2 18287.33} C_VEL
LIN {X 0,Y 385.166,Z 876.11,A -85,B 0,C 180,E1 18284.892,E2 18284.892} C_VEL
LIN {X 0,Y 384.726,Z 885.052,A -85,B 0,C 180,E1 18282.457,E2 18282.457} C_VEL
LIN {X 0,Y 384.578,Z 892.691,A -85,B 0,C 180,E1 18279.818,E2 18279.818} C_VEL
LIN {X 0,Y 384.672,Z 898.431,A -85,B 0,C 180,E1 18277.167,E2 18277.167} C_VEL
LIN {X 0,Y 384.865,Z 902.228,A -85,B 0,C 180,E1 18274.62,E2 18274.62} C_VEL
LIN {X 0,Y 385.024,Z 904.378,A -85,B 0,C 180,E1 18272.084,E2 18272.084} C_VEL
LIN {X 0,Y 385.063,Z 904.926,A -85,B 0,C 180,E1 18269.554,E2 18269.554} C_VEL
LIN {X 0,Y 384.965,Z 903.885,A -85,B 0,C 180,E1 18267.023,E2 18267.023} C_VEL
LIN {X 0,Y 384.772,Z 901.148,A -85,B 0,C 180,E1 18264.414,E2 18264.414} C_VEL
LIN {X 0,Y 384.583,Z 896.655,A -85,B 0,C 180,E1 18261.779,E2 18261.779} C_VEL
LIN {X 0,Y 384.568,Z 890.557,A -85,B 0,C 180,E1 18259.211,E2 18259.211} C_VEL
LIN {X 0,Y 384.825,Z 882.591,A -85,B 0,C 180,E1 18256.63,E2 18256.63} C_VEL
LIN {X 0,Y 385.42,Z 873.199,A -85,B 0,C 180,E1 18254.194,E2 18254.194} C_VEL
LIN {X 0,Y 386.378,Z 862.456,A -85,B 0,C 180,E1 18251.909,E2 18251.909} C_VEL
LIN {X 0,Y 387.669,Z 850.409,A -85,B 0,C 180,E1 18249.781,E2 18249.781} C_VEL
LIN {X 0,Y 389.329,Z 836.465,A -85,B 0,C 180,E1 18247.741,E2 18247.741} C_VEL
LIN {X 0,Y 391.141,Z 821.513,A -85,B 0,C 180,E1 18245.938,E2 18245.938} C_VEL
LIN {X 0,Y 393.077,Z 805.618,A -85,B 0,C 180,E1 18244.379,E2 18244.379} C_VEL
LIN {X 0,Y 394.958,Z 788.774,A -85,B 0,C 180,E1 18243.054,E2 18243.054} C_VEL
LIN {X 0,Y 396.61,Z 772.182,A -85,B 0,C 180,E1 18242.037,E2 18242.037} C_VEL
LIN {X 0,Y 398.117,Z 754.235,A -85,B 0,C 180,E1 18241.219,E2 18241.219} C_VEL
LIN {X 0,Y 399.198,Z 735.51,A -85,B 0,C 180,E1 18240.641,E2 18240.641} C_VEL
LIN {X 0,Y 402.68,Z 565.568,A -85,B 0,C 180,E1 18237.514,E2 18237.514} C_VEL
LIN {X 0,Y 400.044,Z 541.568,A -85,B 0,C 180,E1 18236.75,E2 18236.75} C_VEL
LIN {X 0,Y 404.906,Z 506.061,A -85,B 0,C 180,E1 18232.902,E2 18232.902} C_VEL
LIN {X 0,Y 399.814,Z 490.259,A -85,B 0,C 180,E1 18230.264,E2 18230.264} C_VEL
LIN {X 0,Y 394.432,Z 475.881,A -85,B 0,C 180,E1 18227.533,E2 18227.533} C_VEL
LIN {X 0,Y 388.755,Z 462.301,A -85,B 0,C 180,E1 18224.599,E2 18224.599} C_VEL
LIN {X 0,Y 385.647,Z 454.948,A -85,B 0,C 180,E1 18222.787,E2 18222.787} C_VEL
LIN {X 0,Y 385.627,Z 454.75,A -85,B 0,C 180,E1 18218.863,E2 18218.863} C_VEL
LIN {X 0,Y 385.619,Z 454.757,A -85,B 0,C 180,E1 18214.78,E2 18214.78} C_VEL
LIN {X 0,Y 385.627,Z 454.761,A -85,B 0,C 180,E1 18210.716,E2 18210.716} C_VEL
LIN {X 0,Y 385.621,Z 454.761,A -85,B 0,C 180,E1 18206.651,E2 18206.651} C_VEL
LIN {X 0,Y 385.625,Z 454.756,A -85,B 0,C 180,E1 18202.565,E2 18202.565} C_VEL
LIN {X 0,Y 385.617,Z 454.747,A -85,B 0,C 180,E1 18198.598,E2 18198.598} C_VEL
LIN {X 0,Y 385.615,Z 454.739,A -85,B 0,C 180,E1 18194.567,E2 18194.567} C_VEL
LIN {X 0,Y 385.612,Z 454.749,A -85,B 0,C 180,E1 18190.608,E2 18190.608} C_VEL
LIN {X 0,Y 385.611,Z 454.762,A -85,B 0,C 180,E1 18186.551,E2 18186.551} C_VEL
LIN {X 0,Y 385.611,Z 454.764,A -85,B 0,C 180,E1 18182.526,E2 18182.526} C_VEL
LIN {X 0,Y 385.61,Z 454.752,A -85,B 0,C 180,E1 18178.514,E2 18178.514} C_VEL
LIN {X 0,Y 385.607,Z 454.746,A -85,B 0,C 180,E1 18174.494,E2 18174.494} C_VEL
LIN {X 0,Y 385.608,Z 454.744,A -85,B 0,C 180,E1 18170.447,E2 18170.447} C_VEL
LIN {X 0,Y 385.607,Z 454.746,A -85,B 0,C 180,E1 18166.352,E2 18166.352} C_VEL
LIN {X 0,Y 385.608,Z 454.749,A -85,B 0,C 180,E1 18162.339,E2 18162.339} C_VEL
LIN {X 0,Y 385.613,Z 454.752,A -85,B 0,C 180,E1 18158.395,E2 18158.395} C_VEL
LIN {X 0,Y 385.613,Z 454.762,A -85,B 0,C 180,E1 18154.341,E2 18154.341} C_VEL
LIN {X 0,Y 385.67,Z 455.074,A -85,B 0,C 180,E1 18152.568,E2 18152.568} C_VEL
LIN {X 0,Y 389.892,Z 466.404,A -85,B 0,C 180,E1 18149.485,E2 18149.485} C_VEL
LIN {X 0,Y 394.187,Z 478.843,A -85,B 0,C 180,E1 18146.429,E2 18146.429} C_VEL
LIN {X 0,Y 398.234,Z 492.869,A -85,B 0,C 180,E1 18143.305,E2 18143.305} C_VEL
LIN {X 0,Y 400.131,Z 501.086,A -85,B 0,C 180,E1 18141.622,E2 18141.622} C_VEL
LIN {X 0,Y 396.612,Z 528.546,A -85,B 0,C 180,E1 18137.3,E2 18137.3} C_VEL
LIN {X 0,Y 393.848,Z 553.57,A -85,B 0,C 180,E1 18133.442,E2 18133.442} C_VEL
LIN {X 0,Y 394.799,Z 558.77,A -85,B 0,C 180,E1 18133.178,E2 18133.178} C_VEL
LIN {X 0,Y 399.596,Z 584.613,A -85,B 0,C 180,E1 18132.211,E2 18132.211} C_VEL
LIN {X 0,Y 397.12,Z 680.019,A -85,B 0,C 180,E1 18130.302,E2 18130.302} C_VEL
LIN {X 0,Y 396.474,Z 696.042,A -85,B 0,C 180,E1 18129.711,E2 18129.711} C_VEL
LIN {X 0,Y 395.548,Z 710.568,A -85,B 0,C 180,E1 18128.914,E2 18128.914} C_VEL
LIN {X 0,Y 394.231,Z 725.621,A -85,B 0,C 180,E1 18127.777,E2 18127.777} C_VEL
LIN {X 0,Y 392.871,Z 738.023,A -85,B 0,C 180,E1 18126.55,E2 18126.55} C_VEL
LIN {X 0,Y 391.39,Z 750.222,A -85,B 0,C 180,E1 18125.017,E2 18125.017} C_VEL
LIN {X 0,Y 389.927,Z 761.001,A -85,B 0,C 180,E1 18123.281,E2 18123.281} C_VEL
LIN {X 0,Y 388.671,Z 769.85,A -85,B 0,C 180,E1 18121.481,E2 18121.481} C_VEL
LIN {X 0,Y 387.484,Z 777.835,A -85,B 0,C 180,E1 18119.358,E2 18119.358} C_VEL
LIN {X 0,Y 386.607,Z 783.747,A -85,B 0,C 180,E1 18117.243,E2 18117.243} C_VEL
LIN {X 0,Y 385.937,Z 788.351,A -85,B 0,C 180,E1 18114.815,E2 18114.815} C_VEL
LIN {X 0,Y 385.573,Z 790.73,A -85,B 0,C 180,E1 18112.568,E2 18112.568} C_VEL
LIN {X 0,Y 385.408,Z 791.486,A -85,B 0,C 180,E1 18110.184,E2 18110.184} C_VEL
LIN {X 0,Y 385.427,Z 790.373,A -85,B 0,C 180,E1 18107.812,E2 18107.812} C_VEL
LIN {X 0,Y 385.626,Z 787.775,A -85,B 0,C 180,E1 18105.643,E2 18105.643} C_VEL
LIN {X 0,Y 386.053,Z 783.1,A -85,B 0,C 180,E1 18103.327,E2 18103.327} C_VEL
LIN {X 0,Y 386.71,Z 776.883,A -85,B 0,C 180,E1 18101.181,E2 18101.181} C_VEL
LIN {X 0,Y 387.632,Z 768.578,A -85,B 0,C 180,E1 18099.052,E2 18099.052} C_VEL
LIN {X 0,Y 388.748,Z 758.51,A -85,B 0,C 180,E1 18097.091,E2 18097.091} C_VEL
LIN {X 0,Y 389.727,Z 749.48,A -85,B 0,C 180,E1 18095.684,E2 18095.684} C_VEL
LIN {X 0,Y 389.378,Z 743.966,A -85,B 0,C 180,E1 18094.879,E2 18094.879} C_VEL
LIN {X 0,Y 386.206,Z 733.575,A -85,B 0,C 180,E1 18093.451,E2 18093.451} C_VEL
LIN {X 0,Y 384.768,Z 726.567,A -85,B 0,C 180,E1 18092.663,E2 18092.663} C_VEL
LIN {X 0,Y 384.748,Z 722.79,A -85,B 0,C 180,E1 18092.318,E2 18092.318} C_VEL
LIN {X 0,Y 385.824,Z 708.313,A -85,B 0,C 180,E1 18091.262,E2 18091.262} C_VEL
LIN {X 0,Y 386.683,Z 691.943,A -85,B 0,C 180,E1 18090.416,E2 18090.416} C_VEL
LIN {X 0,Y 387.167,Z 676.158,A -85,B 0,C 180,E1 18089.903,E2 18089.903} C_VEL
LIN {X 0,Y 388.981,Z 582.556,A -85,B 0,C 180,E1 18088.062,E2 18088.062} C_VEL
LIN {X 0,Y 384.115,Z 554.054,A -85,B 0,C 180,E1 18087.128,E2 18087.128} C_VEL
LIN {X 0,Y 386.748,Z 525.865,A -85,B 0,C 180,E1 18082.871,E2 18082.871} C_VEL
LIN {X 0,Y 389.778,Z 498.235,A -85,B 0,C 180,E1 18078.608,E2 18078.608} C_VEL
LIN {X 0,Y 385.431,Z 481.506,A -85,B 0,C 180,E1 18075.379,E2 18075.379} C_VEL
LIN {X 0,Y 380.725,Z 465.643,A -85,B 0,C 180,E1 18072.105,E2 18072.105} C_VEL
LIN {X 0,Y 377.651,Z 455.872,A -85,B 0,C 180,E1 18069.928,E2 18069.928} C_VEL
LIN {X 0,Y 377.622,Z 455.714,A -85,B 0,C 180,E1 18065.992,E2 18065.992} C_VEL
LIN {X 0,Y 377.616,Z 455.748,A -85,B 0,C 180,E1 18062.052,E2 18062.052} C_VEL
LIN {X 0,Y 377.61,Z 455.747,A -85,B 0,C 180,E1 18058.202,E2 18058.202} C_VEL
LIN {X 0,Y 377.612,Z 455.75,A -85,B 0,C 180,E1 18054.12,E2 18054.12} C_VEL
LIN {X 0,Y 377.616,Z 455.759,A -85,B 0,C 180,E1 18050.15,E2 18050.15} C_VEL
LIN {X 0,Y 377.618,Z 455.753,A -85,B 0,C 180,E1 18046.072,E2 18046.072} C_VEL
LIN {X 0,Y 377.618,Z 455.736,A -85,B 0,C 180,E1 18042.06,E2 18042.06} C_VEL
LIN {X 0,Y 377.625,Z 455.757,A -85,B 0,C 180,E1 18037.904,E2 18037.904} C_VEL
LIN {X 0,Y 377.624,Z 455.726,A -85,B 0,C 180,E1 18033.757,E2 18033.757} C_VEL
LIN {X 0,Y 377.631,Z 455.756,A -85,B 0,C 180,E1 18029.678,E2 18029.678} C_VEL
LIN {X 0,Y 377.63,Z 455.723,A -85,B 0,C 180,E1 18025.568,E2 18025.568} C_VEL
LIN {X 0,Y 377.635,Z 455.756,A -85,B 0,C 180,E1 18021.594,E2 18021.594} C_VEL
LIN {X 0,Y 377.633,Z 455.715,A -85,B 0,C 180,E1 18017.568,E2 18017.568} C_VEL
LIN {X 0,Y 377.641,Z 455.754,A -85,B 0,C 180,E1 18013.474,E2 18013.474} C_VEL
LIN {X 0,Y 377.64,Z 455.721,A -85,B 0,C 180,E1 18009.448,E2 18009.448} C_VEL
LIN {X 0,Y 377.645,Z 455.75,A -85,B 0,C 180,E1 18005.317,E2 18005.317} C_VEL
LIN {X 0,Y 377.645,Z 455.727,A -85,B 0,C 180,E1 18001.214,E2 18001.214} C_VEL
LIN {X 0,Y 377.649,Z 455.75,A -85,B 0,C 180,E1 17997.117,E2 17997.117} C_VEL
LIN {X 0,Y 377.651,Z 455.73,A -85,B 0,C 180,E1 17993.005,E2 17993.005} C_VEL
LIN {X 0,Y 377.653,Z 455.752,A -85,B 0,C 180,E1 17989.011,E2 17989.011} C_VEL
LIN {X 0,Y 377.654,Z 455.727,A -85,B 0,C 180,E1 17984.962,E2 17984.962} C_VEL
LIN {X 0,Y 377.661,Z 455.754,A -85,B 0,C 180,E1 17980.835,E2 17980.835} C_VEL
LIN {X 0,Y 377.662,Z 455.747,A -85,B 0,C 180,E1 17976.735,E2 17976.735} C_VEL
LIN {X 0,Y 377.661,Z 455.733,A -85,B 0,C 180,E1 17972.741,E2 17972.741} C_VEL
LIN {X 0,Y 377.667,Z 455.74,A -85,B 0,C 180,E1 17968.742,E2 17968.742} C_VEL
LIN {X 0,Y 377.667,Z 455.743,A -85,B 0,C 180,E1 17964.629,E2 17964.629} C_VEL
LIN {X 0,Y 377.667,Z 455.742,A -85,B 0,C 180,E1 17960.551,E2 17960.551} C_VEL
LIN {X 0,Y 377.673,Z 455.75,A -85,B 0,C 180,E1 17956.502,E2 17956.502} C_VEL
LIN {X 0,Y 377.729,Z 456.069,A -85,B 0,C 180,E1 17954.998,E2 17954.998} C_VEL
LIN {X 0,Y 384.524,Z 474.379,A -85,B 0,C 180,E1 17951.732,E2 17951.732} C_VEL
LIN {X 0,Y 391.679,Z 495.224,A -85,B 0,C 180,E1 17948.4,E2 17948.4} C_VEL
LIN {X 0,Y 395.036,Z 505.639,A -85,B 0,C 180,E1 17946.86,E2 17946.86} C_VEL
LIN {X 0,Y 390.73,Z 541.635,A -85,B 0,C 180,E1 17943.051,E2 17943.051} C_VEL
LIN {X 0,Y 393.453,Z 569.309,A -85,B 0,C 180,E1 17942.299,E2 17942.299} C_VEL
LIN {X 0,Y 390.138,Z 737.021,A -85,B 0,C 180,E1 17939.237,E2 17939.237} C_VEL
LIN {X 0,Y 389.109,Z 755.527,A -85,B 0,C 180,E1 17938.646,E2 17938.646} C_VEL
LIN {X 0,Y 387.719,Z 773.421,A -85,B 0,C 180,E1 17937.806,E2 17937.806} C_VEL
LIN {X 0,Y 386.035,Z 791.251,A -85,B 0,C 180,E1 17936.674,E2 17936.674} C_VEL
LIN {X 0,Y 384.327,Z 807.63,A -85,B 0,C 180,E1 17935.339,E2 17935.339} C_VEL
LIN {X 0,Y 382.512,Z 823.436,A -85,B 0,C 180,E1 17933.738,E2 17933.738} C_VEL
LIN {X 0,Y 380.829,Z 838.298,A -85,B 0,C 180,E1 17931.89,E2 17931.89} C_VEL
LIN {X 0,Y 379.343,Z 851.624,A -85,B 0,C 180,E1 17929.878,E2 17929.878} C_VEL
LIN {X 0,Y 378.159,Z 863.521,A -85,B 0,C 180,E1 17927.702,E2 17927.702} C_VEL
LIN {X 0,Y 377.253,Z 874.658,A -85,B 0,C 180,E1 17925.212,E2 17925.212} C_VEL
LIN {X 0,Y 376.772,Z 883.67,A -85,B 0,C 180,E1 17922.725,E2 17922.725} C_VEL
LIN {X 0,Y 376.614,Z 891.213,A -85,B 0,C 180,E1 17920.092,E2 17920.092} C_VEL
LIN {X 0,Y 376.704,Z 896.891,A -85,B 0,C 180,E1 17917.473,E2 17917.473} C_VEL
LIN {X 0,Y 376.921,Z 900.834,A -85,B 0,C 180,E1 17914.87,E2 17914.87} C_VEL
LIN {X 0,Y 377.094,Z 903.117,A -85,B 0,C 180,E1 17912.28,E2 17912.28} C_VEL
LIN {X 0,Y 377.148,Z 903.788,A -85,B 0,C 180,E1 17909.696,E2 17909.696} C_VEL
LIN {X 0,Y 377.044,Z 902.848,A -85,B 0,C 180,E1 17907.112,E2 17907.112} C_VEL
LIN {X 0,Y 376.838,Z 900.284,A -85,B 0,C 180,E1 17904.519,E2 17904.519} C_VEL
LIN {X 0,Y 376.628,Z 896.087,A -85,B 0,C 180,E1 17901.912,E2 17901.912} C_VEL
LIN {X 0,Y 376.587,Z 890.027,A -85,B 0,C 180,E1 17899.225,E2 17899.225} C_VEL
LIN {X 0,Y 376.847,Z 881.956,A -85,B 0,C 180,E1 17896.498,E2 17896.498} C_VEL
LIN {X 0,Y 377.53,Z 872.021,A -85,B 0,C 180,E1 17893.854,E2 17893.854} C_VEL
LIN {X 0,Y 378.646,Z 860.49,A -85,B 0,C 180,E1 17891.367,E2 17891.367} C_VEL
LIN {X 0,Y 380.188,Z 847.331,A -85,B 0,C 180,E1 17889.043,E2 17889.043} C_VEL
LIN {X 0,Y 382.015,Z 832.991,A -85,B 0,C 180,E1 17886.965,E2 17886.965} C_VEL
LIN {X 0,Y 383.944,Z 818.241,A -85,B 0,C 180,E1 17885.212,E2 17885.212} C_VEL
LIN {X 0,Y 386.014,Z 801.935,A -85,B 0,C 180,E1 17883.635,E2 17883.635} C_VEL
LIN {X 0,Y 387.946,Z 785.349,A -85,B 0,C 180,E1 17882.36,E2 17882.36} C_VEL
LIN {X 0,Y 389.715,Z 767.95,A -85,B 0,C 180,E1 17881.33,E2 17881.33} C_VEL
LIN {X 0,Y 391.223,Z 749.858,A -85,B 0,C 180,E1 17880.551,E2 17880.551} C_VEL
LIN {X 0,Y 392.204,Z 731.285,A -85,B 0,C 180,E1 17880.022,E2 17880.022} C_VEL
LIN {X 0,Y 395.777,Z 566.479,A -85,B 0,C 180,E1 17876.943,E2 17876.943} C_VEL
LIN {X 0,Y 393.059,Z 541.876,A -85,B 0,C 180,E1 17876.146,E2 17876.146} C_VEL
LIN {X 0,Y 397.872,Z 509.073,A -85,B 0,C 180,E1 17872.518,E2 17872.518} C_VEL
LIN {X 0,Y 393.06,Z 494.027,A -85,B 0,C 180,E1 17869.941,E2 17869.941} C_VEL
LIN {X 0,Y 387.973,Z 480.264,A -85,B 0,C 180,E1 17867.263,E2 17867.263} C_VEL
LIN {X 0,Y 382.707,Z 467.43,A -85,B 0,C 180,E1 17864.441,E2 17864.441} C_VEL
LIN {X 0,Y 378.791,Z 458.918,A -85,B 0,C 180,E1 17862.307,E2 17862.307} C_VEL
LIN {X 0,Y 377.698,Z 455.907,A -85,B 0,C 180,E1 17861.482,E2 17861.482} C_VEL
LIN {X 0,Y 377.678,Z 455.754,A -85,B 0,C 180,E1 17857.419,E2 17857.419} C_VEL
LIN {X 0,Y 377.676,Z 455.744,A -85,B 0,C 180,E1 17853.22,E2 17853.22} C_VEL
LIN {X 0,Y 377.677,Z 455.74,A -85,B 0,C 180,E1 17849.116,E2 17849.116} C_VEL
LIN {X 0,Y 377.675,Z 455.742,A -85,B 0,C 180,E1 17845.061,E2 17845.061} C_VEL
LIN {X 0,Y 377.675,Z 455.749,A -85,B 0,C 180,E1 17840.94,E2 17840.94} C_VEL
LIN {X 0,Y 377.676,Z 455.752,A -85,B 0,C 180,E1 17836.772,E2 17836.772} C_VEL
LIN {X 0,Y 377.675,Z 455.751,A -85,B 0,C 180,E1 17832.693,E2 17832.693} C_VEL
LIN {X 0,Y 377.676,Z 455.738,A -85,B 0,C 180,E1 17828.525,E2 17828.525} C_VEL
LIN {X 0,Y 377.67,Z 455.729,A -85,B 0,C 180,E1 17824.555,E2 17824.555} C_VEL
LIN {X 0,Y 377.67,Z 455.734,A -85,B 0,C 180,E1 17820.455,E2 17820.455} C_VEL
LIN {X 0,Y 377.672,Z 455.747,A -85,B 0,C 180,E1 17816.357,E2 17816.357} C_VEL
LIN {X 0,Y 377.671,Z 455.752,A -85,B 0,C 180,E1 17812.24,E2 17812.24} C_VEL
LIN {X 0,Y 377.671,Z 455.753,A -85,B 0,C 180,E1 17808.237,E2 17808.237} C_VEL
LIN {X 0,Y 377.671,Z 455.754,A -85,B 0,C 180,E1 17804.175,E2 17804.175} C_VEL
LIN {X 0,Y 377.672,Z 455.751,A -85,B 0,C 180,E1 17800.023,E2 17800.023} C_VEL
LIN {X 0,Y 377.671,Z 455.742,A -85,B 0,C 180,E1 17795.939,E2 17795.939} C_VEL
LIN {X 0,Y 377.717,Z 456.059,A -85,B 0,C 180,E1 17793.814,E2 17793.814} C_VEL
LIN {X 0,Y 381.896,Z 466.955,A -85,B 0,C 180,E1 17790.673,E2 17790.673} C_VEL
LIN {X 0,Y 386.304,Z 479.504,A -85,B 0,C 180,E1 17787.427,E2 17787.427} C_VEL
LIN {X 0,Y 390.331,Z 492.97,A -85,B 0,C 180,E1 17784.293,E2 17784.293} C_VEL
LIN {X 0,Y 392.984,Z 503.725,A -85,B 0,C 180,E1 17781.996,E2 17781.996} C_VEL
LIN {X 0,Y 389.387,Z 530.436,A -85,B 0,C 180,E1 17777.719,E2 17777.719} C_VEL
LIN {X 0,Y 386.711,Z 553.906,A -85,B 0,C 180,E1 17774.068,E2 17774.068} C_VEL
LIN {X 0,Y 391.937,Z 580.786,A -85,B 0,C 180,E1 17772.959,E2 17772.959} C_VEL
LIN {X 0,Y 392.675,Z 586.592,A -85,B 0,C 180,E1 17772.769,E2 17772.769} C_VEL
LIN {X 0,Y 390.096,Z 680.646,A -85,B 0,C 180,E1 17770.852,E2 17770.852} C_VEL
LIN {X 0,Y 389.414,Z 696.68,A -85,B 0,C 180,E1 17770.252,E2 17770.252} C_VEL
LIN {X 0,Y 388.443,Z 711.173,A -85,B 0,C 180,E1 17769.447,E2 17769.447} C_VEL
LIN {X 0,Y 387.068,Z 726.019,A -85,B 0,C 180,E1 17768.313,E2 17768.313} C_VEL
LIN {X 0,Y 385.67,Z 738.184,A -85,B 0,C 180,E1 17767.106,E2 17767.106} C_VEL
LIN {X 0,Y 384.02,Z 750.877,A -85,B 0,C 180,E1 17765.494,E2 17765.494} C_VEL
LIN {X 0,Y 382.49,Z 761.491,A -85,B 0,C 180,E1 17763.769,E2 17763.769} C_VEL
LIN {X 0,Y 381.054,Z 770.9,A -85,B 0,C 180,E1 17761.83,E2 17761.83} C_VEL
LIN {X 0,Y 379.777,Z 778.897,A -85,B 0,C 180,E1 17759.667,E2 17759.667} C_VEL
LIN {X 0,Y 378.829,Z 784.836,A -85,B 0,C 180,E1 17757.509,E2 17757.509} C_VEL
LIN {X 0,Y 378.092,Z 789.458,A -85,B 0,C 180,E1 17755.031,E2 17755.031} C_VEL
LIN {X 0,Y 377.688,Z 791.875,A -85,B 0,C 180,E1 17752.737,E2 17752.737} C_VEL
LIN {X 0,Y 377.498,Z 792.663,A -85,B 0,C 180,E1 17750.302,E2 17750.302} C_VEL
LIN {X 0,Y 377.506,Z 791.605,A -85,B 0,C 180,E1 17747.893,E2 17747.893} C_VEL
LIN {X 0,Y 377.729,Z 788.796,A -85,B 0,C 180,E1 17745.506,E2 17745.506} C_VEL
LIN {X 0,Y 378.188,Z 784.063,A -85,B 0,C 180,E1 17743.142,E2 17743.142} C_VEL
LIN {X 0,Y 378.887,Z 777.78,A -85,B 0,C 180,E1 17740.953,E2 17740.953} C_VEL
LIN {X 0,Y 379.867,Z 769.418,A -85,B 0,C 180,E1 17738.781,E2 17738.781} C_VEL
LIN {X 0,Y 381.048,Z 759.289,A -85,B 0,C 180,E1 17736.781,E2 17736.781} C_VEL
LIN {X 0,Y 382.267,Z 748.463,A -85,B 0,C 180,E1 17735.102,E2 17735.102} C_VEL
LIN {X 0,Y 383.537,Z 736.112,A -85,B 0,C 180,E1 17733.587,E2 17733.587} C_VEL
LIN {X 0,Y 384.748,Z 722.79,A -85,B 0,C 180,E1 17732.318,E2 17732.318} C_VEL
LIN {X 0,Y 384.341,Z 716.091,A -85,B 0,C 180,E1 17731.733,E2 17731.733} C_VEL
LIN {X 0,Y 380.767,Z 702.843,A -85,B 0,C 180,E1 17730.597,E2 17730.597} C_VEL
LIN {X 0,Y 379.349,Z 694.772,A -85,B 0,C 180,E1 17730.082,E2 17730.082} C_VEL
LIN {X 0,Y 379.307,Z 691.592,A -85,B 0,C 180,E1 17729.938,E2 17729.938} C_VEL
LIN {X 0,Y 379.813,Z 674.697,A -85,B 0,C 180,E1 17729.406,E2 17729.406} C_VEL
LIN {X 0,Y 381.667,Z 583.67,A -85,B 0,C 180,E1 17727.593,E2 17727.593} C_VEL
LIN {X 0,Y 376.615,Z 553.796,A -85,B 0,C 180,E1 17726.595,E2 17726.595} C_VEL
LIN {X 0,Y 379.42,Z 525.769,A -85,B 0,C 180,E1 17722.276,E2 17722.276} C_VEL
LIN {X 0,Y 382.288,Z 500.478,A -85,B 0,C 180,E1 17718.305,E2 17718.305} C_VEL
LIN {X 0,Y 377.872,Z 483.538,A -85,B 0,C 180,E1 17714.971,E2 17714.971} C_VEL
LIN {X 0,Y 373.1,Z 467.402,A -85,B 0,C 180,E1 17711.565,E2 17711.565} C_VEL
LIN {X 0,Y 369.714,Z 456.842,A -85,B 0,C 180,E1 17709.126,E2 17709.126} C_VEL
LIN {X 0,Y 369.704,Z 456.71,A -85,B 0,C 180,E1 17705.216,E2 17705.216} C_VEL
LIN {X 0,Y 369.712,Z 456.733,A -85,B 0,C 180,E1 17701.192,E2 17701.192} C_VEL
LIN {X 0,Y 369.704,Z 456.733,A -85,B 0,C 180,E1 17697.07,E2 17697.07} C_VEL
LIN {X 0,Y 369.7,Z 456.728,A -85,B 0,C 180,E1 17692.924,E2 17692.924} C_VEL
LIN {X 0,Y 369.712,Z 456.73,A -85,B 0,C 180,E1 17688.915,E2 17688.915} C_VEL
LIN {X 0,Y 369.716,Z 456.746,A -85,B 0,C 180,E1 17684.882,E2 17684.882} C_VEL
LIN {X 0,Y 369.717,Z 456.718,A -85,B 0,C 180,E1 17680.779,E2 17680.779} C_VEL
LIN {X 0,Y 369.719,Z 456.736,A -85,B 0,C 180,E1 17676.703,E2 17676.703} C_VEL
LIN {X 0,Y 369.717,Z 456.725,A -85,B 0,C 180,E1 17672.56,E2 17672.56} C_VEL
LIN {X 0,Y 369.732,Z 456.73,A -85,B 0,C 180,E1 17668.598,E2 17668.598} C_VEL
LIN {X 0,Y 369.723,Z 456.721,A -85,B 0,C 180,E1 17664.442,E2 17664.442} C_VEL
LIN {X 0,Y 369.732,Z 456.732,A -85,B 0,C 180,E1 17660.418,E2 17660.418} C_VEL
LIN {X 0,Y 369.725,Z 456.711,A -85,B 0,C 180,E1 17656.251,E2 17656.251} C_VEL
LIN {X 0,Y 369.737,Z 456.737,A -85,B 0,C 180,E1 17652.336,E2 17652.336} C_VEL
LIN {X 0,Y 369.737,Z 456.702,A -85,B 0,C 180,E1 17648.207,E2 17648.207} C_VEL
LIN {X 0,Y 369.739,Z 456.739,A -85,B 0,C 180,E1 17644.187,E2 17644.187} C_VEL
LIN {X 0,Y 369.738,Z 456.702,A -85,B 0,C 180,E1 17640,E2 17640} C_VEL
LIN {X 0,Y 369.739,Z 456.741,A -85,B 0,C 180,E1 17635.969,E2 17635.969} C_VEL
LIN {X 0,Y 369.742,Z 456.707,A -85,B 0,C 180,E1 17631.917,E2 17631.917} C_VEL
LIN {X 0,Y 369.744,Z 456.739,A -85,B 0,C 180,E1 17627.824,E2 17627.824} C_VEL
LIN {X 0,Y 369.744,Z 456.719,A -85,B 0,C 180,E1 17623.738,E2 17623.738} C_VEL
LIN {X 0,Y 369.744,Z 456.725,A -85,B 0,C 180,E1 17619.584,E2 17619.584} C_VEL
LIN {X 0,Y 369.746,Z 456.74,A -85,B 0,C 180,E1 17615.56,E2 17615.56} C_VEL
LIN {X 0,Y 369.749,Z 456.735,A -85,B 0,C 180,E1 17611.404,E2 17611.404} C_VEL
LIN {X 0,Y 369.742,Z 456.731,A -85,B 0,C 180,E1 17607.247,E2 17607.247} C_VEL
LIN {X 0,Y 369.741,Z 456.734,A -85,B 0,C 180,E1 17603.106,E2 17603.106} C_VEL
LIN {X 0,Y 369.748,Z 456.742,A -85,B 0,C 180,E1 17598.979,E2 17598.979} C_VEL
LIN {X 0,Y 369.778,Z 456.975,A -85,B 0,C 180,E1 17595.849,E2 17595.849} C_VEL
LIN {X 0,Y 376.734,Z 475.669,A -85,B 0,C 180,E1 17592.386,E2 17592.386} C_VEL
LIN {X 0,Y 383.706,Z 495.895,A -85,B 0,C 180,E1 17589.057,E2 17589.057} C_VEL
LIN {X 0,Y 387.572,Z 508.643,A -85,B 0,C 180,E1 17587.134,E2 17587.134} C_VEL
LIN {X 0,Y 383.412,Z 542.031,A -85,B 0,C 180,E1 17583.547,E2 17583.547} C_VEL
LIN {X 0,Y 386.17,Z 570.135,A -85,B 0,C 180,E1 17582.778,E2 17582.778} C_VEL
LIN {X 0,Y 382.719,Z 736.436,A -85,B 0,C 180,E1 17579.689,E2 17579.689} C_VEL
LIN {X 0,Y 381.66,Z 754.918,A -85,B 0,C 180,E1 17579.087,E2 17579.087} C_VEL
LIN {X 0,Y 380.234,Z 772.513,A -85,B 0,C 180,E1 17578.248,E2 17578.248} C_VEL
LIN {X 0,Y 378.476,Z 790.442,A -85,B 0,C 180,E1 17577.091,E2 17577.091} C_VEL
LIN {X 0,Y 376.681,Z 806.912,A -85,B 0,C 180,E1 17575.722,E2 17575.722} C_VEL
LIN {X 0,Y 374.79,Z 822.684,A -85,B 0,C 180,E1 17574.09,E2 17574.09} C_VEL
LIN {X 0,Y 373.032,Z 837.512,A -85,B 0,C 180,E1 17572.206,E2 17572.206} C_VEL
LIN {X 0,Y 371.398,Z 851.535,A -85,B 0,C 180,E1 17570.023,E2 17570.023} C_VEL
LIN {X 0,Y 370.173,Z 863.417,A -85,B 0,C 180,E1 17567.772,E2 17567.772} C_VEL
LIN {X 0,Y 369.301,Z 873.795,A -85,B 0,C 180,E1 17565.387,E2 17565.387} C_VEL
LIN {X 0,Y 368.803,Z 882.776,A -85,B 0,C 180,E1 17562.845,E2 17562.845} C_VEL
LIN {X 0,Y 368.648,Z 890.27,A -85,B 0,C 180,E1 17560.154,E2 17560.154} C_VEL
LIN {X 0,Y 368.769,Z 896.169,A -85,B 0,C 180,E1 17557.322,E2 17557.322} C_VEL
LIN {X 0,Y 369.008,Z 899.953,A -85,B 0,C 180,E1 17554.663,E2 17554.663} C_VEL
LIN {X 0,Y 369.196,Z 902.072,A -85,B 0,C 180,E1 17552.018,E2 17552.018} C_VEL
LIN {X 0,Y 369.232,Z 902.567,A -85,B 0,C 180,E1 17549.38,E2 17549.38} C_VEL
LIN {X 0,Y 369.096,Z 901.451,A -85,B 0,C 180,E1 17546.739,E2 17546.739} C_VEL
LIN {X 0,Y 368.858,Z 898.725,A -85,B 0,C 180,E1 17544.088,E2 17544.088} C_VEL
LIN {X 0,Y 368.631,Z 894.345,A -85,B 0,C 180,E1 17541.421,E2 17541.421} C_VEL
LIN {X 0,Y 368.631,Z 887.806,A -85,B 0,C 180,E1 17538.58,E2 17538.58} C_VEL
LIN {X 0,Y 368.958,Z 879.727,A -85,B 0,C 180,E1 17535.884,E2 17535.884} C_VEL
LIN {X 0,Y 369.71,Z 870.222,A -85,B 0,C 180,E1 17533.342,E2 17533.342} C_VEL
LIN {X 0,Y 370.943,Z 858.545,A -85,B 0,C 180,E1 17530.802,E2 17530.802} C_VEL
LIN {X 0,Y 372.506,Z 846.177,A -85,B 0,C 180,E1 17528.59,E2 17528.59} C_VEL
LIN {X 0,Y 374.372,Z 832.388,A -85,B 0,C 180,E1 17526.551,E2 17526.551} C_VEL
LIN {X 0,Y 376.414,Z 817.719,A -85,B 0,C 180,E1 17524.765,E2 17524.765} C_VEL
LIN {X 0,Y 378.603,Z 801.477,A -85,B 0,C 180,E1 17523.154,E2 17523.154} C_VEL
LIN {X 0,Y 380.622,Z 785.179,A -85,B 0,C 180,E1 17521.867,E2 17521.867} C_VEL
LIN {X 0,Y 382.549,Z 767.456,A -85,B 0,C 180,E1 17520.788,E2 17520.788} C_VEL
LIN {X 0,Y 384.135,Z 749.256,A -85,B 0,C 180,E1 17519.99,E2 17519.99} C_VEL
LIN {X 0,Y 385.161,Z 730.741,A -85,B 0,C 180,E1 17519.454,E2 17519.454} C_VEL
LIN {X 0,Y 388.93,Z 567.456,A -85,B 0,C 180,E1 17516.351,E2 17516.351} C_VEL
LIN {X 0,Y 386.157,Z 541.912,A -85,B 0,C 180,E1 17515.49,E2 17515.49} C_VEL
LIN {X 0,Y 390.832,Z 512.092,A -85,B 0,C 180,E1 17512.122,E2 17512.122} C_VEL
LIN {X 0,Y 386.049,Z 496.946,A -85,B 0,C 180,E1 17509.452,E2 17509.452} C_VEL
LIN {X 0,Y 380.583,Z 482.234,A -85,B 0,C 180,E1 17506.477,E2 17506.477} C_VEL
LIN {X 0,Y 375.175,Z 469.122,A -85,B 0,C 180,E1 17503.439,E2 17503.439} C_VEL
LIN {X 0,Y 370.889,Z 459.962,A -85,B 0,C 180,E1 17500.989,E2 17500.989} C_VEL
LIN {X 0,Y 369.764,Z 456.861,A -85,B 0,C 180,E1 17500.058,E2 17500.058} C_VEL
LIN {X 0,Y 369.741,Z 456.726,A -85,B 0,C 180,E1 17495.931,E2 17495.931} C_VEL
LIN {X 0,Y 369.743,Z 456.724,A -85,B 0,C 180,E1 17491.824,E2 17491.824} C_VEL
LIN {X 0,Y 369.745,Z 456.722,A -85,B 0,C 180,E1 17487.718,E2 17487.718} C_VEL
LIN {X 0,Y 369.742,Z 456.72,A -85,B 0,C 180,E1 17483.549,E2 17483.549} C_VEL
LIN {X 0,Y 369.739,Z 456.719,A -85,B 0,C 180,E1 17479.428,E2 17479.428} C_VEL
LIN {X 0,Y 369.743,Z 456.72,A -85,B 0,C 180,E1 17475.367,E2 17475.367} C_VEL
LIN {X 0,Y 369.738,Z 456.734,A -85,B 0,C 180,E1 17471.227,E2 17471.227} C_VEL
LIN {X 0,Y 369.74,Z 456.743,A -85,B 0,C 180,E1 17467.048,E2 17467.048} C_VEL
LIN {X 0,Y 369.736,Z 456.734,A -85,B 0,C 180,E1 17462.945,E2 17462.945} C_VEL
LIN {X 0,Y 369.74,Z 456.721,A -85,B 0,C 180,E1 17458.915,E2 17458.915} C_VEL
LIN {X 0,Y 369.733,Z 456.72,A -85,B 0,C 180,E1 17454.724,E2 17454.724} C_VEL
LIN {X 0,Y 369.733,Z 456.721,A -85,B 0,C 180,E1 17450.662,E2 17450.662} C_VEL
LIN {X 0,Y 369.733,Z 456.723,A -85,B 0,C 180,E1 17446.551,E2 17446.551} C_VEL
LIN {X 0,Y 369.734,Z 456.725,A -85,B 0,C 180,E1 17442.532,E2 17442.532} C_VEL
LIN {X 0,Y 369.737,Z 456.728,A -85,B 0,C 180,E1 17438.421,E2 17438.421} C_VEL
LIN {X 0,Y 369.787,Z 457.016,A -85,B 0,C 180,E1 17435.174,E2 17435.174} C_VEL
LIN {X 0,Y 374.14,Z 468.129,A -85,B 0,C 180,E1 17431.769,E2 17431.769} C_VEL
LIN {X 0,Y 378.484,Z 480.307,A -85,B 0,C 180,E1 17428.461,E2 17428.461} C_VEL
LIN {X 0,Y 382.507,Z 493.421,A -85,B 0,C 180,E1 17425.26,E2 17425.26} C_VEL
LIN {X 0,Y 385.842,Z 506.752,A -85,B 0,C 180,E1 17422.32,E2 17422.32} C_VEL
LIN {X 0,Y 381.988,Z 533.764,A -85,B 0,C 180,E1 17417.926,E2 17417.926} C_VEL
LIN {X 0,Y 379.586,Z 553.669,A -85,B 0,C 180,E1 17414.774,E2 17414.774} C_VEL
LIN {X 0,Y 384.755,Z 580.166,A -85,B 0,C 180,E1 17413.629,E2 17413.629} C_VEL
LIN {X 0,Y 385.82,Z 587.638,A -85,B 0,C 180,E1 17413.364,E2 17413.364} C_VEL
LIN {X 0,Y 383.111,Z 681.309,A -85,B 0,C 180,E1 17411.421,E2 17411.421} C_VEL
LIN {X 0,Y 382.39,Z 697.307,A -85,B 0,C 180,E1 17410.813,E2 17410.813} C_VEL
LIN {X 0,Y 381.332,Z 712.213,A -85,B 0,C 180,E1 17409.97,E2 17409.97} C_VEL
LIN {X 0,Y 379.85,Z 727.327,A -85,B 0,C 180,E1 17408.79,E2 17408.79} C_VEL
LIN {X 0,Y 378.235,Z 740.4,A -85,B 0,C 180,E1 17407.445,E2 17407.445} C_VEL
LIN {X 0,Y 376.544,Z 752.62,A -85,B 0,C 180,E1 17405.838,E2 17405.838} C_VEL
LIN {X 0,Y 374.802,Z 763.85,A -85,B 0,C 180,E1 17403.936,E2 17403.936} C_VEL
LIN {X 0,Y 373.343,Z 772.695,A -85,B 0,C 180,E1 17402.023,E2 17402.023} C_VEL
LIN {X 0,Y 371.963,Z 780.762,A -85,B 0,C 180,E1 17399.744,E2 17399.744} C_VEL
LIN {X 0,Y 370.927,Z 786.661,A -85,B 0,C 180,E1 17397.448,E2 17397.448} C_VEL
LIN {X 0,Y 370.214,Z 790.816,A -85,B 0,C 180,E1 17395.088,E2 17395.088} C_VEL
LIN {X 0,Y 369.763,Z 793.228,A -85,B 0,C 180,E1 17392.58,E2 17392.58} C_VEL
LIN {X 0,Y 369.579,Z 793.812,A -85,B 0,C 180,E1 17390.152,E2 17390.152} C_VEL
LIN {X 0,Y 369.603,Z 792.569,A -85,B 0,C 180,E1 17387.637,E2 17387.637} C_VEL
LIN {X 0,Y 369.833,Z 789.813,A -85,B 0,C 180,E1 17385.364,E2 17385.364} C_VEL
LIN {X 0,Y 370.334,Z 784.969,A -85,B 0,C 180,E1 17382.925,E2 17382.925} C_VEL
LIN {X 0,Y 371.07,Z 778.674,A -85,B 0,C 180,E1 17380.715,E2 17380.715} C_VEL
LIN {X 0,Y 372.084,Z 770.471,A -85,B 0,C 180,E1 17378.548,E2 17378.548} C_VEL
LIN {X 0,Y 373.251,Z 760.932,A -85,B 0,C 180,E1 17376.614,E2 17376.614} C_VEL
LIN {X 0,Y 374.522,Z 750.299,A -85,B 0,C 180,E1 17374.9,E2 17374.9} C_VEL
LIN {X 0,Y 375.905,Z 737.454,A -85,B 0,C 180,E1 17373.278,E2 17373.278} C_VEL
LIN {X 0,Y 377.179,Z 724.172,A -85,B 0,C 180,E1 17371.975,E2 17371.975} C_VEL
LIN {X 0,Y 378.289,Z 710.022,A -85,B 0,C 180,E1 17370.908,E2 17370.908} C_VEL
LIN {X 0,Y 379.162,Z 694.593,A -85,B 0,C 180,E1 17370.071,E2 17370.071} C_VEL
LIN {X 0,Y 379.307,Z 691.592,A -85,B 0,C 180,E1 17369.938,E2 17369.938} C_VEL
LIN {X 0,Y 378.724,Z 684.149,A -85,B 0,C 180,E1 17369.612,E2 17369.612} C_VEL
LIN {X 0,Y 373.582,Z 665.446,A -85,B 0,C 180,E1 17368.799,E2 17368.799} C_VEL
LIN {X 0,Y 372.799,Z 657.858,A -85,B 0,C 180,E1 17368.585,E2 17368.585} C_VEL
LIN {X 0,Y 374.333,Z 584.604,A -85,B 0,C 180,E1 17367.108,E2 17367.108} C_VEL
LIN {X 0,Y 369.147,Z 553.528,A -85,B 0,C 180,E1 17366.039,E2 17366.039} C_VEL
LIN {X 0,Y 372.123,Z 525.656,A -85,B 0,C 180,E1 17361.657,E2 17361.657} C_VEL
LIN {X 0,Y 374.77,Z 502.7,A -85,B 0,C 180,E1 17357.989,E2 17357.989} C_VEL
LIN {X 0,Y 370.333,Z 485.603,A -85,B 0,C 180,E1 17354.551,E2 17354.551} C_VEL
LIN {X 0,Y 365.694,Z 469.993,A -85,B 0,C 180,E1 17351.178,E2 17351.178} C_VEL
LIN {X 0,Y 361.758,Z 457.861,A -85,B 0,C 180,E1 17348.322,E2 17348.322} C_VEL
LIN {X 0,Y 361.738,Z 457.725,A -85,B 0,C 180,E1 17344.281,E2 17344.281} C_VEL
LIN {X 0,Y 361.734,Z 457.738,A -85,B 0,C 180,E1 17340.163,E2 17340.163} C_VEL
LIN {X 0,Y 361.737,Z 457.736,A -85,B 0,C 180,E1 17336.019,E2 17336.019} C_VEL
LIN {X 0,Y 361.738,Z 457.728,A -85,B 0,C 180,E1 17331.947,E2 17331.947} C_VEL
LIN {X 0,Y 361.738,Z 457.714,A -85,B 0,C 180,E1 17328.018,E2 17328.018} C_VEL
LIN {X 0,Y 361.745,Z 457.736,A -85,B 0,C 180,E1 17323.829,E2 17323.829} C_VEL
LIN {X 0,Y 361.748,Z 457.724,A -85,B 0,C 180,E1 17319.791,E2 17319.791} C_VEL
LIN {X 0,Y 361.749,Z 457.714,A -85,B 0,C 180,E1 17315.648,E2 17315.648} C_VEL
LIN {X 0,Y 361.752,Z 457.729,A -85,B 0,C 180,E1 17311.647,E2 17311.647} C_VEL
LIN {X 0,Y 361.753,Z 457.71,A -85,B 0,C 180,E1 17307.668,E2 17307.668} C_VEL
LIN {X 0,Y 361.756,Z 457.726,A -85,B 0,C 180,E1 17303.627,E2 17303.627} C_VEL
LIN {X 0,Y 361.759,Z 457.714,A -85,B 0,C 180,E1 17299.526,E2 17299.526} C_VEL
LIN {X 0,Y 361.76,Z 457.719,A -85,B 0,C 180,E1 17295.387,E2 17295.387} C_VEL
LIN {X 0,Y 361.764,Z 457.723,A -85,B 0,C 180,E1 17291.317,E2 17291.317} C_VEL
LIN {X 0,Y 361.767,Z 457.708,A -85,B 0,C 180,E1 17287.145,E2 17287.145} C_VEL
LIN {X 0,Y 361.772,Z 457.727,A -85,B 0,C 180,E1 17283.01,E2 17283.01} C_VEL
LIN {X 0,Y 361.775,Z 457.704,A -85,B 0,C 180,E1 17278.892,E2 17278.892} C_VEL
LIN {X 0,Y 361.782,Z 457.728,A -85,B 0,C 180,E1 17274.768,E2 17274.768} C_VEL
LIN {X 0,Y 361.779,Z 457.709,A -85,B 0,C 180,E1 17270.776,E2 17270.776} C_VEL
LIN {X 0,Y 361.786,Z 457.719,A -85,B 0,C 180,E1 17266.611,E2 17266.611} C_VEL
LIN {X 0,Y 361.792,Z 457.726,A -85,B 0,C 180,E1 17262.451,E2 17262.451} C_VEL
LIN {X 0,Y 361.8,Z 457.706,A -85,B 0,C 180,E1 17258.265,E2 17258.265} C_VEL
LIN {X 0,Y 361.8,Z 457.716,A -85,B 0,C 180,E1 17254.11,E2 17254.11} C_VEL
LIN {X 0,Y 361.811,Z 457.727,A -85,B 0,C 180,E1 17249.988,E2 17249.988} C_VEL
LIN {X 0,Y 361.807,Z 457.73,A -85,B 0,C 180,E1 17245.876,E2 17245.876} C_VEL
LIN {X 0,Y 361.809,Z 457.726,A -85,B 0,C 180,E1 17241.706,E2 17241.706} C_VEL
LIN {X 0,Y 361.807,Z 457.719,A -85,B 0,C 180,E1 17237.55,E2 17237.55} C_VEL
LIN {X 0,Y 361.857,Z 458.122,A -85,B 0,C 180,E1 17236.672,E2 17236.672} C_VEL
LIN {X 0,Y 368.947,Z 476.943,A -85,B 0,C 180,E1 17233.073,E2 17233.073} C_VEL
LIN {X 0,Y 375.734,Z 496.566,A -85,B 0,C 180,E1 17229.731,E2 17229.731} C_VEL
LIN {X 0,Y 380.205,Z 510.87,A -85,B 0,C 180,E1 17227.503,E2 17227.503} C_VEL
LIN {X 0,Y 376.096,Z 541.684,A -85,B 0,C 180,E1 17224.099,E2 17224.099} C_VEL
LIN {X 0,Y 378.882,Z 570.99,A -85,B 0,C 180,E1 17223.264,E2 17223.264} C_VEL
LIN {X 0,Y 375.316,Z 735.754,A -85,B 0,C 180,E1 17220.155,E2 17220.155} C_VEL
LIN {X 0,Y 374.235,Z 754.223,A -85,B 0,C 180,E1 17219.545,E2 17219.545} C_VEL
LIN {X 0,Y 372.691,Z 772.469,A -85,B 0,C 180,E1 17218.657,E2 17218.657} C_VEL
LIN {X 0,Y 370.941,Z 789.617,A -85,B 0,C 180,E1 17217.525,E2 17217.525} C_VEL
LIN {X 0,Y 369.052,Z 806.195,A -85,B 0,C 180,E1 17216.121,E2 17216.121} C_VEL
LIN {X 0,Y 367.083,Z 821.932,A -85,B 0,C 180,E1 17214.458,E2 17214.458} C_VEL
LIN {X 0,Y 365.25,Z 836.726,A -85,B 0,C 180,E1 17212.535,E2 17212.535} C_VEL
LIN {X 0,Y 363.543,Z 850.705,A -85,B 0,C 180,E1 17210.305,E2 17210.305} C_VEL
LIN {X 0,Y 362.26,Z 862.548,A -85,B 0,C 180,E1 17208.007,E2 17208.007} C_VEL
LIN {X 0,Y 361.353,Z 872.89,A -85,B 0,C 180,E1 17205.569,E2 17205.569} C_VEL
LIN {X 0,Y 360.837,Z 881.84,A -85,B 0,C 180,E1 17202.971,E2 17202.971} C_VEL
LIN {X 0,Y 360.684,Z 889.307,A -85,B 0,C 180,E1 17200.22,E2 17200.22} C_VEL
LIN {X 0,Y 360.823,Z 895.167,A -85,B 0,C 180,E1 17197.324,E2 17197.324} C_VEL
LIN {X 0,Y 361.091,Z 898.95,A -85,B 0,C 180,E1 17194.558,E2 17194.558} C_VEL
LIN {X 0,Y 361.287,Z 900.952,A -85,B 0,C 180,E1 17191.903,E2 17191.903} C_VEL
LIN {X 0,Y 361.315,Z 901.37,A -85,B 0,C 180,E1 17189.207,E2 17189.207} C_VEL
LIN {X 0,Y 361.154,Z 900.17,A -85,B 0,C 180,E1 17186.508,E2 17186.508} C_VEL
LIN {X 0,Y 360.878,Z 897.352,A -85,B 0,C 180,E1 17183.797,E2 17183.797} C_VEL
LIN {X 0,Y 360.647,Z 892.883,A -85,B 0,C 180,E1 17181.069,E2 17181.069} C_VEL
LIN {X 0,Y 360.658,Z 886.68,A -85,B 0,C 180,E1 17178.324,E2 17178.324} C_VEL
LIN {X 0,Y 361.023,Z 878.6,A -85,B 0,C 180,E1 17175.567,E2 17175.567} C_VEL
LIN {X 0,Y 361.848,Z 869.029,A -85,B 0,C 180,E1 17172.953,E2 17172.953} C_VEL
LIN {X 0,Y 363.178,Z 857.405,A -85,B 0,C 180,E1 17170.374,E2 17170.374} C_VEL
LIN {X 0,Y 364.855,Z 845.028,A -85,B 0,C 180,E1 17168.118,E2 17168.118} C_VEL
LIN {X 0,Y 366.842,Z 831.27,A -85,B 0,C 180,E1 17166.039,E2 17166.039} C_VEL
LIN {X 0,Y 369.041,Z 816.493,A -85,B 0,C 180,E1 17164.207,E2 17164.207} C_VEL
LIN {X 0,Y 371.334,Z 800.369,A -85,B 0,C 180,E1 17162.585,E2 17162.585} C_VEL
LIN {X 0,Y 373.464,Z 784.022,A -85,B 0,C 180,E1 17161.278,E2 17161.278} C_VEL
LIN {X 0,Y 375.497,Z 766.162,A -85,B 0,C 180,E1 17160.185,E2 17160.185} C_VEL
LIN {X 0,Y 377.116,Z 748.251,A -85,B 0,C 180,E1 17159.394,E2 17159.394} C_VEL
LIN {X 0,Y 378.171,Z 729.759,A -85,B 0,C 180,E1 17158.855,E2 17158.855} C_VEL
LIN {X 0,Y 382.117,Z 568.327,A -85,B 0,C 180,E1 17155.735,E2 17155.735} C_VEL
LIN {X 0,Y 379.301,Z 542.246,A -85,B 0,C 180,E1 17154.832,E2 17154.832} C_VEL
LIN {X 0,Y 383.734,Z 514.742,A -85,B 0,C 180,E1 17151.655,E2 17151.655} C_VEL
LIN {X 0,Y 379.058,Z 500.049,A -85,B 0,C 180,E1 17148.972,E2 17148.972} C_VEL
LIN {X 0,Y 374.135,Z 486.609,A -85,B 0,C 180,E1 17146.183,E2 17146.183} C_VEL
LIN {X 0,Y 368.817,Z 473.627,A -85,B 0,C 180,E1 17143.092,E2 17143.092} C_VEL
LIN {X 0,Y 364.817,Z 464.933,A -85,B 0,C 180,E1 17140.714,E2 17140.714} C_VEL
LIN {X 0,Y 363.237,Z 461.396,A -85,B 0,C 180,E1 17139.688,E2 17139.688} C_VEL
LIN {X 0,Y 361.826,Z 457.868,A -85,B 0,C 180,E1 17138.553,E2 17138.553} C_VEL
LIN {X 0,Y 361.805,Z 457.729,A -85,B 0,C 180,E1 17134.316,E2 17134.316} C_VEL
LIN {X 0,Y 361.807,Z 457.732,A -85,B 0,C 180,E1 17130.12,E2 17130.12} C_VEL
LIN {X 0,Y 361.807,Z 457.73,A -85,B 0,C 180,E1 17125.889,E2 17125.889} C_VEL
LIN {X 0,Y 361.81,Z 457.73,A -85,B 0,C 180,E1 17121.734,E2 17121.734} C_VEL
LIN {X 0,Y 361.805,Z 457.726,A -85,B 0,C 180,E1 17117.531,E2 17117.531} C_VEL
LIN {X 0,Y 361.804,Z 457.712,A -85,B 0,C 180,E1 17113.403,E2 17113.403} C_VEL
LIN {X 0,Y 361.799,Z 457.706,A -85,B 0,C 180,E1 17109.223,E2 17109.223} C_VEL
LIN {X 0,Y 361.801,Z 457.707,A -85,B 0,C 180,E1 17105.232,E2 17105.232} C_VEL
LIN {X 0,Y 361.804,Z 457.718,A -85,B 0,C 180,E1 17101.108,E2 17101.108} C_VEL
LIN {X 0,Y 361.8,Z 457.73,A -85,B 0,C 180,E1 17096.99,E2 17096.99} C_VEL
LIN {X 0,Y 361.802,Z 457.731,A -85,B 0,C 180,E1 17092.798,E2 17092.798} C_VEL
LIN {X 0,Y 361.798,Z 457.727,A -85,B 0,C 180,E1 17088.684,E2 17088.684} C_VEL
LIN {X 0,Y 361.796,Z 457.73,A -85,B 0,C 180,E1 17084.45,E2 17084.45} C_VEL
LIN {X 0,Y 361.795,Z 457.732,A -85,B 0,C 180,E1 17080.296,E2 17080.296} C_VEL
LIN {X 0,Y 361.847,Z 458.011,A -85,B 0,C 180,E1 17076.648,E2 17076.648} C_VEL
LIN {X 0,Y 366.277,Z 468.969,A -85,B 0,C 180,E1 17073.054,E2 17073.054} C_VEL
LIN {X 0,Y 370.724,Z 481.242,A -85,B 0,C 180,E1 17069.532,E2 17069.532} C_VEL
LIN {X 0,Y 374.701,Z 493.91,A -85,B 0,C 180,E1 17066.287,E2 17066.287} C_VEL
LIN {X 0,Y 378.116,Z 507.039,A -85,B 0,C 180,E1 17063.247,E2 17063.247} C_VEL
LIN {X 0,Y 378.636,Z 510.118,A -85,B 0,C 180,E1 17062.601,E2 17062.601} C_VEL
LIN {X 0,Y 374.595,Z 537.18,A -85,B 0,C 180,E1 17058.133,E2 17058.133} C_VEL
LIN {X 0,Y 372.501,Z 553.245,A -85,B 0,C 180,E1 17055.527,E2 17055.527} C_VEL
LIN {X 0,Y 376.419,Z 572.745,A -85,B 0,C 180,E1 17054.612,E2 17054.612} C_VEL
LIN {X 0,Y 379.027,Z 588.799,A -85,B 0,C 180,E1 17053.985,E2 17053.985} C_VEL
LIN {X 0,Y 376.169,Z 681.942,A -85,B 0,C 180,E1 17052.014,E2 17052.014} C_VEL
LIN {X 0,Y 375.406,Z 697.911,A -85,B 0,C 180,E1 17051.397,E2 17051.397} C_VEL
LIN {X 0,Y 374.336,Z 712.425,A -85,B 0,C 180,E1 17050.571,E2 17050.571} C_VEL
LIN {X 0,Y 372.843,Z 726.952,A -85,B 0,C 180,E1 17049.435,E2 17049.435} C_VEL
LIN {X 0,Y 371.163,Z 740.168,A -85,B 0,C 180,E1 17048.089,E2 17048.089} C_VEL
LIN {X 0,Y 369.374,Z 752.37,A -85,B 0,C 180,E1 17046.49,E2 17046.49} C_VEL
LIN {X 0,Y 367.728,Z 762.607,A -85,B 0,C 180,E1 17044.8,E2 17044.8} C_VEL
LIN {X 0,Y 365.986,Z 772.547,A -85,B 0,C 180,E1 17042.706,E2 17042.706} C_VEL
LIN {X 0,Y 364.546,Z 780.409,A -85,B 0,C 180,E1 17040.545,E2 17040.545} C_VEL
LIN {X 0,Y 363.379,Z 786.663,A -85,B 0,C 180,E1 17038.246,E2 17038.246} C_VEL
LIN {X 0,Y 362.515,Z 791.193,A -85,B 0,C 180,E1 17035.835,E2 17035.835} C_VEL
LIN {X 0,Y 361.985,Z 793.936,A -85,B 0,C 180,E1 17033.437,E2 17033.437} C_VEL
LIN {X 0,Y 361.697,Z 794.992,A -85,B 0,C 180,E1 17030.875,E2 17030.875} C_VEL
LIN {X 0,Y 361.657,Z 794.298,A -85,B 0,C 180,E1 17028.371,E2 17028.371} C_VEL
LIN {X 0,Y 361.842,Z 791.781,A -85,B 0,C 180,E1 17025.876,E2 17025.876} C_VEL
LIN {X 0,Y 362.257,Z 787.819,A -85,B 0,C 180,E1 17023.568,E2 17023.568} C_VEL
LIN {X 0,Y 363.001,Z 781.582,A -85,B 0,C 180,E1 17021.117,E2 17021.117} C_VEL
LIN {X 0,Y 363.931,Z 774.353,A -85,B 0,C 180,E1 17019.009,E2 17019.009} C_VEL
LIN {X 0,Y 365.134,Z 765.038,A -85,B 0,C 180,E1 17016.92,E2 17016.92} C_VEL
LIN {X 0,Y 366.418,Z 754.869,A -85,B 0,C 180,E1 17015.127,E2 17015.127} C_VEL
LIN {X 0,Y 367.844,Z 742.703,A -85,B 0,C 180,E1 17013.428,E2 17013.428} C_VEL
LIN {X 0,Y 369.197,Z 729.749,A -85,B 0,C 180,E1 17012.017,E2 17012.017} C_VEL
LIN {X 0,Y 370.426,Z 715.93,A -85,B 0,C 180,E1 17010.846,E2 17010.846} C_VEL
LIN {X 0,Y 371.455,Z 700.589,A -85,B 0,C 180,E1 17009.891,E2 17009.891} C_VEL
LIN {X 0,Y 372.147,Z 685.191,A -85,B 0,C 180,E1 17009.23,E2 17009.23} C_VEL
LIN {X 0,Y 372.667,Z 663.319,A -85,B 0,C 180,E1 17008.698,E2 17008.698} C_VEL
LIN {X 0,Y 372.799,Z 657.858,A -85,B 0,C 180,E1 17008.585,E2 17008.585} C_VEL
LIN {X 0,Y 372.067,Z 650.257,A -85,B 0,C 180,E1 17008.367,E2 17008.367} C_VEL
LIN {X 0,Y 366.841,Z 630.315,A -85,B 0,C 180,E1 17007.569,E2 17007.569} C_VEL
LIN {X 0,Y 366.313,Z 623.78,A -85,B 0,C 180,E1 17007.388,E2 17007.388} C_VEL
LIN {X 0,Y 367.046,Z 585.671,A -85,B 0,C 180,E1 17006.608,E2 17006.608} C_VEL
LIN {X 0,Y 361.709,Z 553.479,A -85,B 0,C 180,E1 17005.481,E2 17005.481} C_VEL
LIN {X 0,Y 364.854,Z 525.512,A -85,B 0,C 180,E1 17001.013,E2 17001.013} C_VEL
LIN {X 0,Y 367.343,Z 505.275,A -85,B 0,C 180,E1 16997.731,E2 16997.731} C_VEL
LIN {X 0,Y 363.098,Z 488.764,A -85,B 0,C 180,E1 16994.344,E2 16994.344} C_VEL
LIN {X 0,Y 358.567,Z 473.388,A -85,B 0,C 180,E1 16990.958,E2 16990.958} C_VEL
LIN {X 0,Y 353.866,Z 458.849,A -85,B 0,C 180,E1 16987.464,E2 16987.464} C_VEL
LIN {X 0,Y 353.832,Z 458.723,A -85,B 0,C 180,E1 16983.248,E2 16983.248} C_VEL
LIN {X 0,Y 353.823,Z 458.718,A -85,B 0,C 180,E1 16979.048,E2 16979.048} C_VEL
LIN {X 0,Y 353.824,Z 458.721,A -85,B 0,C 180,E1 16974.994,E2 16974.994} C_VEL
LIN {X 0,Y 353.834,Z 458.723,A -85,B 0,C 180,E1 16970.938,E2 16970.938} C_VEL
LIN {X 0,Y 353.826,Z 458.703,A -85,B 0,C 180,E1 16966.809,E2 16966.809} C_VEL
LIN {X 0,Y 353.828,Z 458.704,A -85,B 0,C 180,E1 16962.704,E2 16962.704} C_VEL
LIN {X 0,Y 353.836,Z 458.722,A -85,B 0,C 180,E1 16958.646,E2 16958.646} C_VEL
LIN {X 0,Y 353.835,Z 458.685,A -85,B 0,C 180,E1 16954.61,E2 16954.61} C_VEL
LIN {X 0,Y 353.835,Z 458.722,A -85,B 0,C 180,E1 16950.386,E2 16950.386} C_VEL
LIN {X 0,Y 353.833,Z 458.68,A -85,B 0,C 180,E1 16946.337,E2 16946.337} C_VEL
LIN {X 0,Y 353.841,Z 458.721,A -85,B 0,C 180,E1 16942.25,E2 16942.25} C_VEL
LIN {X 0,Y 353.834,Z 458.678,A -85,B 0,C 180,E1 16938.11,E2 16938.11} C_VEL
LIN {X 0,Y 353.844,Z 458.719,A -85,B 0,C 180,E1 16934.065,E2 16934.065} C_VEL
LIN {X 0,Y 353.837,Z 458.687,A -85,B 0,C 180,E1 16929.926,E2 16929.926} C_VEL
LIN {X 0,Y 353.842,Z 458.713,A -85,B 0,C 180,E1 16925.839,E2 16925.839} C_VEL
LIN {X 0,Y 353.842,Z 458.697,A -85,B 0,C 180,E1 16921.782,E2 16921.782} C_VEL
LIN {X 0,Y 353.847,Z 458.709,A -85,B 0,C 180,E1 16917.733,E2 16917.733} C_VEL
LIN {X 0,Y 353.843,Z 458.699,A -85,B 0,C 180,E1 16913.51,E2 16913.51} C_VEL
LIN {X 0,Y 353.844,Z 458.717,A -85,B 0,C 180,E1 16909.417,E2 16909.417} C_VEL
LIN {X 0,Y 353.842,Z 458.691,A -85,B 0,C 180,E1 16905.267,E2 16905.267} C_VEL
LIN {X 0,Y 353.846,Z 458.72,A -85,B 0,C 180,E1 16901.037,E2 16901.037} C_VEL
LIN {X 0,Y 353.847,Z 458.712,A -85,B 0,C 180,E1 16896.873,E2 16896.873} C_VEL
LIN {X 0,Y 353.846,Z 458.698,A -85,B 0,C 180,E1 16892.757,E2 16892.757} C_VEL
LIN {X 0,Y 353.851,Z 458.704,A -85,B 0,C 180,E1 16888.578,E2 16888.578} C_VEL
LIN {X 0,Y 353.852,Z 458.706,A -85,B 0,C 180,E1 16884.403,E2 16884.403} C_VEL
LIN {X 0,Y 353.856,Z 458.707,A -85,B 0,C 180,E1 16880.226,E2 16880.226} C_VEL
LIN {X 0,Y 353.908,Z 458.981,A -85,B 0,C 180,E1 16877.623,E2 16877.623} C_VEL
LIN {X 0,Y 360.223,Z 475.725,A -85,B 0,C 180,E1 16874.265,E2 16874.265} C_VEL
LIN {X 0,Y 366.556,Z 493.629,A -85,B 0,C 180,E1 16871.044,E2 16871.044} C_VEL
LIN {X 0,Y 372.835,Z 513.067,A -85,B 0,C 180,E1 16867.889,E2 16867.889} C_VEL
LIN {X 0,Y 368.823,Z 541.945,A -85,B 0,C 180,E1 16864.637,E2 16864.637} C_VEL
LIN {X 0,Y 371.62,Z 571.821,A -85,B 0,C 180,E1 16863.767,E2 16863.767} C_VEL
LIN {X 0,Y 367.91,Z 735.136,A -85,B 0,C 180,E1 16860.629,E2 16860.629} C_VEL
LIN {X 0,Y 366.799,Z 753.589,A -85,B 0,C 180,E1 16860.008,E2 16860.008} C_VEL
LIN {X 0,Y 365.218,Z 771.552,A -85,B 0,C 180,E1 16859.119,E2 16859.119} C_VEL
LIN {X 0,Y 363.418,Z 788.659,A -85,B 0,C 180,E1 16857.975,E2 16857.975} C_VEL
LIN {X 0,Y 361.437,Z 805.377,A -85,B 0,C 180,E1 16856.537,E2 16856.537} C_VEL
LIN {X 0,Y 359.393,Z 821.142,A -85,B 0,C 180,E1 16854.841,E2 16854.841} C_VEL
LIN {X 0,Y 357.481,Z 835.937,A -85,B 0,C 180,E1 16852.879,E2 16852.879} C_VEL
LIN {X 0,Y 355.793,Z 849.134,A -85,B 0,C 180,E1 16850.738,E2 16850.738} C_VEL
LIN {X 0,Y 354.354,Z 861.678,A -85,B 0,C 180,E1 16848.253,E2 16848.253} C_VEL
LIN {X 0,Y 353.406,Z 871.985,A -85,B 0,C 180,E1 16845.76,E2 16845.76} C_VEL
LIN {X 0,Y 352.852,Z 881.389,A -85,B 0,C 180,E1 16842.936,E2 16842.936} C_VEL
LIN {X 0,Y 352.722,Z 888.706,A -85,B 0,C 180,E1 16840.123,E2 16840.123} C_VEL
LIN {X 0,Y 352.879,Z 894.146,A -85,B 0,C 180,E1 16837.326,E2 16837.326} C_VEL
LIN {X 0,Y 353.168,Z 897.829,A -85,B 0,C 180,E1 16834.547,E2 16834.547} C_VEL
LIN {X 0,Y 353.378,Z 899.825,A -85,B 0,C 180,E1 16831.784,E2 16831.784} C_VEL
LIN {X 0,Y 353.394,Z 900.174,A -85,B 0,C 180,E1 16829.028,E2 16829.028} C_VEL
LIN {X 0,Y 353.204,Z 898.895,A -85,B 0,C 180,E1 16826.267,E2 16826.267} C_VEL
LIN {X 0,Y 352.895,Z 895.989,A -85,B 0,C 180,E1 16823.493,E2 16823.493} C_VEL
LIN {X 0,Y 352.657,Z 891.279,A -85,B 0,C 180,E1 16820.628,E2 16820.628} C_VEL
LIN {X 0,Y 352.713,Z 884.681,A -85,B 0,C 180,E1 16817.725,E2 16817.725} C_VEL
LIN {X 0,Y 353.184,Z 876.285,A -85,B 0,C 180,E1 16814.876,E2 16814.876} C_VEL
LIN {X 0,Y 354.215,Z 865.949,A -85,B 0,C 180,E1 16812.081,E2 16812.081} C_VEL
LIN {X 0,Y 355.658,Z 854.696,A -85,B 0,C 180,E1 16809.599,E2 16809.599} C_VEL
LIN {X 0,Y 357.613,Z 841.562,A -85,B 0,C 180,E1 16807.218,E2 16807.218} C_VEL
LIN {X 0,Y 359.818,Z 827.285,A -85,B 0,C 180,E1 16805.103,E2 16805.103} C_VEL
LIN {X 0,Y 362.222,Z 811.972,A -85,B 0,C 180,E1 16803.261,E2 16803.261} C_VEL
LIN {X 0,Y 364.603,Z 795.651,A -85,B 0,C 180,E1 16801.679,E2 16801.679} C_VEL
LIN {X 0,Y 366.962,Z 777.94,A -85,B 0,C 180,E1 16800.336,E2 16800.336} C_VEL
LIN {X 0,Y 368.871,Z 760.994,A -85,B 0,C 180,E1 16799.364,E2 16799.364} C_VEL
LIN {X 0,Y 370.478,Z 742.866,A -85,B 0,C 180,E1 16798.623,E2 16798.623} C_VEL
LIN {X 0,Y 371.396,Z 723.956,A -85,B 0,C 180,E1 16798.127,E2 16798.127} C_VEL
LIN {X 0,Y 375.395,Z 569.278,A -85,B 0,C 180,E1 16795.09,E2 16795.09} C_VEL
LIN {X 0,Y 372.516,Z 542.35,A -85,B 0,C 180,E1 16794.129,E2 16794.129} C_VEL
LIN {X 0,Y 376.715,Z 517.694,A -85,B 0,C 180,E1 16791.217,E2 16791.217} C_VEL
LIN {X 0,Y 372.012,Z 502.768,A -85,B 0,C 180,E1 16788.405,E2 16788.405} C_VEL
LIN {X 0,Y 366.822,Z 488.653,A -85,B 0,C 180,E1 16785.35,E2 16785.35} C_VEL
LIN {X 0,Y 361.38,Z 475.445,A -85,B 0,C 180,E1 16782.033,E2 16782.033} C_VEL
LIN {X 0,Y 357.224,Z 466.499,A -85,B 0,C 180,E1 16779.42,E2 16779.42} C_VEL
LIN {X 0,Y 355.187,Z 462.217,A -85,B 0,C 180,E1 16778.06,E2 16778.06} C_VEL
LIN {X 0,Y 353.885,Z 458.864,A -85,B 0,C 180,E1 16776.91,E2 16776.91} C_VEL
LIN {X 0,Y 353.865,Z 458.702,A -85,B 0,C 180,E1 16772.647,E2 16772.647} C_VEL
LIN {X 0,Y 353.873,Z 458.697,A -85,B 0,C 180,E1 16768.512,E2 16768.512} C_VEL
LIN {X 0,Y 353.865,Z 458.697,A -85,B 0,C 180,E1 16764.364,E2 16764.364} C_VEL
LIN {X 0,Y 353.866,Z 458.699,A -85,B 0,C 180,E1 16760.164,E2 16760.164} C_VEL
LIN {X 0,Y 353.869,Z 458.704,A -85,B 0,C 180,E1 16755.907,E2 16755.907} C_VEL
LIN {X 0,Y 353.866,Z 458.718,A -85,B 0,C 180,E1 16751.738,E2 16751.738} C_VEL
LIN {X 0,Y 353.872,Z 458.716,A -85,B 0,C 180,E1 16747.468,E2 16747.468} C_VEL
LIN {X 0,Y 353.862,Z 458.705,A -85,B 0,C 180,E1 16743.239,E2 16743.239} C_VEL
LIN {X 0,Y 353.865,Z 458.696,A -85,B 0,C 180,E1 16739.028,E2 16739.028} C_VEL
LIN {X 0,Y 353.856,Z 458.696,A -85,B 0,C 180,E1 16734.812,E2 16734.812} C_VEL
LIN {X 0,Y 353.857,Z 458.697,A -85,B 0,C 180,E1 16730.731,E2 16730.731} C_VEL
LIN {X 0,Y 353.857,Z 458.7,A -85,B 0,C 180,E1 16726.602,E2 16726.602} C_VEL
LIN {X 0,Y 353.854,Z 458.702,A -85,B 0,C 180,E1 16722.401,E2 16722.401} C_VEL
LIN {X 0,Y 353.89,Z 458.953,A -85,B 0,C 180,E1 16718.298,E2 16718.298} C_VEL
LIN {X 0,Y 357.241,Z 467.15,A -85,B 0,C 180,E1 16715.353,E2 16715.353} C_VEL
LIN {X 0,Y 361.217,Z 477.333,A -85,B 0,C 180,E1 16712.108,E2 16712.108} C_VEL
LIN {X 0,Y 365.187,Z 488.865,A -85,B 0,C 180,E1 16708.837,E2 16708.837} C_VEL
LIN {X 0,Y 369.039,Z 501.983,A -85,B 0,C 180,E1 16705.51,E2 16705.51} C_VEL
LIN {X 0,Y 371.598,Z 512.682,A -85,B 0,C 180,E1 16703.048,E2 16703.048} C_VEL
LIN {X 0,Y 367.599,Z 538.081,A -85,B 0,C 180,E1 16698.77,E2 16698.77} C_VEL
LIN {X 0,Y 365.522,Z 552.92,A -85,B 0,C 180,E1 16696.314,E2 16696.314} C_VEL
LIN {X 0,Y 366.441,Z 558.002,A -85,B 0,C 180,E1 16696.018,E2 16696.018} C_VEL
LIN {X 0,Y 371.804,Z 585.835,A -85,B 0,C 180,E1 16694.781,E2 16694.781} C_VEL
LIN {X 0,Y 372.28,Z 590.591,A -85,B 0,C 180,E1 16694.62,E2 16694.62} C_VEL
LIN {X 0,Y 369.307,Z 682.66,A -85,B 0,C 180,E1 16692.637,E2 16692.637} C_VEL
LIN {X 0,Y 368.495,Z 698.724,A -85,B 0,C 180,E1 16692.005,E2 16692.005} C_VEL
LIN {X 0,Y 367.293,Z 713.859,A -85,B 0,C 180,E1 16691.119,E2 16691.119} C_VEL
LIN {X 0,Y 365.657,Z 728.764,A -85,B 0,C 180,E1 16689.916,E2 16689.916} C_VEL
LIN {X 0,Y 363.927,Z 741.426,A -85,B 0,C 180,E1 16688.584,E2 16688.584} C_VEL
LIN {X 0,Y 361.999,Z 753.779,A -85,B 0,C 180,E1 16686.923,E2 16686.923} C_VEL
LIN {X 0,Y 360.137,Z 764.541,A -85,B 0,C 180,E1 16685.078,E2 16685.078} C_VEL
LIN {X 0,Y 358.331,Z 774.237,A -85,B 0,C 180,E1 16682.964,E2 16682.964} C_VEL
LIN {X 0,Y 356.732,Z 782.333,A -85,B 0,C 180,E1 16680.63,E2 16680.63} C_VEL
LIN {X 0,Y 355.54,Z 788.273,A -85,B 0,C 180,E1 16678.329,E2 16678.329} C_VEL
LIN {X 0,Y 354.598,Z 792.831,A -85,B 0,C 180,E1 16675.736,E2 16675.736} C_VEL
LIN {X 0,Y 354.056,Z 795.332,A -85,B 0,C 180,E1 16673.288,E2 16673.288} C_VEL
LIN {X 0,Y 353.767,Z 796.193,A -85,B 0,C 180,E1 16670.515,E2 16670.515} C_VEL
LIN {X 0,Y 353.752,Z 795.131,A -85,B 0,C 180,E1 16667.943,E2 16667.943} C_VEL
LIN {X 0,Y 353.994,Z 792.348,A -85,B 0,C 180,E1 16665.397,E2 16665.397} C_VEL
LIN {X 0,Y 354.514,Z 787.652,A -85,B 0,C 180,E1 16662.874,E2 16662.874} C_VEL
LIN {X 0,Y 355.313,Z 781.463,A -85,B 0,C 180,E1 16660.539,E2 16660.539} C_VEL
LIN {X 0,Y 356.425,Z 773.192,A -85,B 0,C 180,E1 16658.225,E2 16658.225} C_VEL
LIN {X 0,Y 357.654,Z 764.109,A -85,B 0,C 180,E1 16656.259,E2 16656.259} C_VEL
LIN {X 0,Y 359.15,Z 752.686,A -85,B 0,C 180,E1 16654.311,E2 16654.311} C_VEL
LIN {X 0,Y 360.653,Z 739.952,A -85,B 0,C 180,E1 16652.622,E2 16652.622} C_VEL
LIN {X 0,Y 362.04,Z 726.886,A -85,B 0,C 180,E1 16651.264,E2 16651.264} C_VEL
LIN {X 0,Y 363.324,Z 711.905,A -85,B 0,C 180,E1 16650.079,E2 16650.079} C_VEL
LIN {X 0,Y 364.28,Z 696.691,A -85,B 0,C 180,E1 16649.208,E2 16649.208} C_VEL
LIN {X 0,Y 364.927,Z 680.587,A -85,B 0,C 180,E1 16648.597,E2 16648.597} C_VEL
LIN {X 0,Y 366.313,Z 623.78,A -85,B 0,C 180,E1 16647.388,E2 16647.388} C_VEL
LIN {X 0,Y 365.6,Z 616.174,A -85,B 0,C 180,E1 16647.168,E2 16647.168} C_VEL
LIN {X 0,Y 360.443,Z 596.225,A -85,B 0,C 180,E1 16646.348,E2 16646.348} C_VEL
LIN {X 0,Y 359.937,Z 589.687,A -85,B 0,C 180,E1 16646.165,E2 16646.165} C_VEL
LIN {X 0,Y 359.406,Z 584.423,A -85,B 0,C 180,E1 16646.007,E2 16646.007} C_VEL
LIN {X 0,Y 354.294,Z 553.356,A -85,B 0,C 180,E1 16644.891,E2 16644.891} C_VEL
LIN {X 0,Y 357.617,Z 525.341,A -85,B 0,C 180,E1 16640.342,E2 16640.342} C_VEL
LIN {X 0,Y 359.86,Z 507.559,A -85,B 0,C 180,E1 16637.402,E2 16637.402} C_VEL
LIN {X 0,Y 355.725,Z 491.343,A -85,B 0,C 180,E1 16634.006,E2 16634.006} C_VEL
LIN {X 0,Y 351.128,Z 475.738,A -85,B 0,C 180,E1 16630.485,E2 16630.485} C_VEL
LIN {X 0,Y 346.54,Z 461.996,A -85,B 0,C 180,E1 16627.165,E2 16627.165} C_VEL
LIN {X 0,Y 345.87,Z 459.782,A -85,B 0,C 180,E1 16626.488,E2 16626.488} C_VEL
LIN {X 0,Y 345.858,Z 459.703,A -85,B 0,C 180,E1 16622.207,E2 16622.207} C_VEL
LIN {X 0,Y 345.858,Z 459.699,A -85,B 0,C 180,E1 16618.059,E2 16618.059} C_VEL
LIN {X 0,Y 345.863,Z 459.698,A -85,B 0,C 180,E1 16613.861,E2 16613.861} C_VEL
LIN {X 0,Y 345.868,Z 459.712,A -85,B 0,C 180,E1 16609.747,E2 16609.747} C_VEL
LIN {X 0,Y 345.878,Z 459.708,A -85,B 0,C 180,E1 16605.564,E2 16605.564} C_VEL
LIN {X 0,Y 345.881,Z 459.682,A -85,B 0,C 180,E1 16601.452,E2 16601.452} C_VEL
LIN {X 0,Y 345.888,Z 459.712,A -85,B 0,C 180,E1 16597.35,E2 16597.35} C_VEL
LIN {X 0,Y 345.903,Z 459.68,A -85,B 0,C 180,E1 16593.042,E2 16593.042} C_VEL
LIN {X 0,Y 345.919,Z 459.698,A -85,B 0,C 180,E1 16588.859,E2 16588.859} C_VEL
LIN {X 0,Y 345.911,Z 459.681,A -85,B 0,C 180,E1 16584.597,E2 16584.597} C_VEL
LIN {X 0,Y 345.916,Z 459.698,A -85,B 0,C 180,E1 16580.472,E2 16580.472} C_VEL
LIN {X 0,Y 345.909,Z 459.672,A -85,B 0,C 180,E1 16576.283,E2 16576.283} C_VEL
LIN {X 0,Y 345.911,Z 459.704,A -85,B 0,C 180,E1 16572.182,E2 16572.182} C_VEL
LIN {X 0,Y 345.902,Z 459.668,A -85,B 0,C 180,E1 16567.976,E2 16567.976} C_VEL
LIN {X 0,Y 345.904,Z 459.706,A -85,B 0,C 180,E1 16563.812,E2 16563.812} C_VEL
LIN {X 0,Y 345.9,Z 459.669,A -85,B 0,C 180,E1 16559.669,E2 16559.669} C_VEL
LIN {X 0,Y 345.903,Z 459.708,A -85,B 0,C 180,E1 16555.524,E2 16555.524} C_VEL
LIN {X 0,Y 345.899,Z 459.677,A -85,B 0,C 180,E1 16551.338,E2 16551.338} C_VEL
LIN {X 0,Y 345.903,Z 459.707,A -85,B 0,C 180,E1 16547.14,E2 16547.14} C_VEL
LIN {X 0,Y 345.904,Z 459.701,A -85,B 0,C 180,E1 16542.852,E2 16542.852} C_VEL
LIN {X 0,Y 345.91,Z 459.683,A -85,B 0,C 180,E1 16538.553,E2 16538.553} C_VEL
LIN {X 0,Y 345.916,Z 459.696,A -85,B 0,C 180,E1 16534.306,E2 16534.306} C_VEL
LIN {X 0,Y 345.927,Z 459.707,A -85,B 0,C 180,E1 16530.126,E2 16530.126} C_VEL
LIN {X 0,Y 345.93,Z 459.708,A -85,B 0,C 180,E1 16525.894,E2 16525.894} C_VEL
LIN {X 0,Y 345.932,Z 459.7,A -85,B 0,C 180,E1 16521.562,E2 16521.562} C_VEL
LIN {X 0,Y 345.947,Z 459.906,A -85,B 0,C 180,E1 16518.619,E2 16518.619} C_VEL
LIN {X 0,Y 352.236,Z 476.402,A -85,B 0,C 180,E1 16515.139,E2 16515.139} C_VEL
LIN {X 0,Y 358.819,Z 494.95,A -85,B 0,C 180,E1 16511.687,E2 16511.687} C_VEL
LIN {X 0,Y 365.419,Z 515.492,A -85,B 0,C 180,E1 16508.253,E2 16508.253} C_VEL
LIN {X 0,Y 361.561,Z 542.188,A -85,B 0,C 180,E1 16505.188,E2 16505.188} C_VEL
LIN {X 0,Y 364.385,Z 572.641,A -85,B 0,C 180,E1 16504.291,E2 16504.291} C_VEL
LIN {X 0,Y 360.532,Z 734.518,A -85,B 0,C 180,E1 16501.123,E2 16501.123} C_VEL
LIN {X 0,Y 359.389,Z 752.956,A -85,B 0,C 180,E1 16500.49,E2 16500.49} C_VEL
LIN {X 0,Y 357.706,Z 771.307,A -85,B 0,C 180,E1 16499.562,E2 16499.562} C_VEL
LIN {X 0,Y 355.784,Z 788.809,A -85,B 0,C 180,E1 16498.356,E2 16498.356} C_VEL
LIN {X 0,Y 353.736,Z 805.34,A -85,B 0,C 180,E1 16496.889,E2 16496.889} C_VEL
LIN {X 0,Y 351.665,Z 820.67,A -85,B 0,C 180,E1 16495.191,E2 16495.191} C_VEL
LIN {X 0,Y 349.647,Z 835.588,A -85,B 0,C 180,E1 16493.154,E2 16493.154} C_VEL
LIN {X 0,Y 347.842,Z 849.144,A -85,B 0,C 180,E1 16490.882,E2 16490.882} C_VEL
LIN {X 0,Y 346.454,Z 860.796,A -85,B 0,C 180,E1 16488.51,E2 16488.51} C_VEL
LIN {X 0,Y 345.464,Z 871.079,A -85,B 0,C 180,E1 16485.96,E2 16485.96} C_VEL
LIN {X 0,Y 344.886,Z 880.445,A -85,B 0,C 180,E1 16483.07,E2 16483.07} C_VEL
LIN {X 0,Y 344.758,Z 887.725,A -85,B 0,C 180,E1 16480.19,E2 16480.19} C_VEL
LIN {X 0,Y 344.936,Z 893.122,A -85,B 0,C 180,E1 16477.328,E2 16477.328} C_VEL
LIN {X 0,Y 345.248,Z 896.757,A -85,B 0,C 180,E1 16474.485,E2 16474.485} C_VEL
LIN {X 0,Y 345.469,Z 898.696,A -85,B 0,C 180,E1 16471.659,E2 16471.659} C_VEL
LIN {X 0,Y 345.477,Z 899.009,A -85,B 0,C 180,E1 16469.005,E2 16469.005} C_VEL
LIN {X 0,Y 345.266,Z 897.749,A -85,B 0,C 180,E1 16466.181,E2 16466.181} C_VEL
LIN {X 0,Y 344.925,Z 894.853,A -85,B 0,C 180,E1 16463.342,E2 16463.342} C_VEL
LIN {X 0,Y 344.678,Z 890.294,A -85,B 0,C 180,E1 16460.483,E2 16460.483} C_VEL
LIN {X 0,Y 344.731,Z 883.988,A -85,B 0,C 180,E1 16457.606,E2 16457.606} C_VEL
LIN {X 0,Y 345.234,Z 875.665,A -85,B 0,C 180,E1 16454.671,E2 16454.671} C_VEL
LIN {X 0,Y 346.342,Z 865.293,A -85,B 0,C 180,E1 16451.767,E2 16451.767} C_VEL
LIN {X 0,Y 347.954,Z 853.63,A -85,B 0,C 180,E1 16449.126,E2 16449.126} C_VEL
LIN {X 0,Y 350.041,Z 840.498,A -85,B 0,C 180,E1 16446.696,E2 16446.696} C_VEL
LIN {X 0,Y 352.386,Z 826.212,A -85,B 0,C 180,E1 16444.541,E2 16444.541} C_VEL
LIN {X 0,Y 354.934,Z 810.88,A -85,B 0,C 180,E1 16442.666,E2 16442.666} C_VEL
LIN {X 0,Y 357.447,Z 794.552,A -85,B 0,C 180,E1 16441.059,E2 16441.059} C_VEL
LIN {X 0,Y 359.89,Z 777.178,A -85,B 0,C 180,E1 16439.719,E2 16439.719} C_VEL
LIN {X 0,Y 361.94,Z 759.894,A -85,B 0,C 180,E1 16438.712,E2 16438.712} C_VEL
LIN {X 0,Y 363.613,Z 741.766,A -85,B 0,C 180,E1 16437.964,E2 16437.964} C_VEL
LIN {X 0,Y 364.548,Z 722.906,A -85,B 0,C 180,E1 16437.467,E2 16437.467} C_VEL
LIN {X 0,Y 368.731,Z 570.263,A -85,B 0,C 180,E1 16434.421,E2 16434.421} C_VEL
LIN {X 0,Y 365.812,Z 542.469,A -85,B 0,C 180,E1 16433.394,E2 16433.394} C_VEL
LIN {X 0,Y 369.691,Z 520.549,A -85,B 0,C 180,E1 16430.738,E2 16430.738} C_VEL
LIN {X 0,Y 365.281,Z 506.461,A -85,B 0,C 180,E1 16428.001,E2 16428.001} C_VEL
LIN {X 0,Y 360.413,Z 493.054,A -85,B 0,C 180,E1 16425.025,E2 16425.025} C_VEL
LIN {X 0,Y 355.302,Z 480.415,A -85,B 0,C 180,E1 16421.778,E2 16421.778} C_VEL
LIN {X 0,Y 351.295,Z 471.699,A -85,B 0,C 180,E1 16419.187,E2 16419.187} C_VEL
LIN {X 0,Y 349.265,Z 467.404,A -85,B 0,C 180,E1 16417.78,E2 16417.78} C_VEL
LIN {X 0,Y 347.626,Z 463.732,A -85,B 0,C 180,E1 16416.54,E2 16416.54} C_VEL
LIN {X 0,Y 345.943,Z 459.868,A -85,B 0,C 180,E1 16415.077,E2 16415.077} C_VEL
LIN {X 0,Y 345.931,Z 459.7,A -85,B 0,C 180,E1 16410.77,E2 16410.77} C_VEL
LIN {X 0,Y 345.926,Z 459.701,A -85,B 0,C 180,E1 16406.616,E2 16406.616} C_VEL
LIN {X 0,Y 345.931,Z 459.701,A -85,B 0,C 180,E1 16402.249,E2 16402.249} C_VEL
LIN {X 0,Y 345.927,Z 459.694,A -85,B 0,C 180,E1 16398.015,E2 16398.015} C_VEL
LIN {X 0,Y 345.928,Z 459.684,A -85,B 0,C 180,E1 16393.71,E2 16393.71} C_VEL
LIN {X 0,Y 345.924,Z 459.681,A -85,B 0,C 180,E1 16389.483,E2 16389.483} C_VEL
LIN {X 0,Y 345.923,Z 459.684,A -85,B 0,C 180,E1 16385.307,E2 16385.307} C_VEL
LIN {X 0,Y 345.923,Z 459.692,A -85,B 0,C 180,E1 16380.993,E2 16380.993} C_VEL
LIN {X 0,Y 345.917,Z 459.704,A -85,B 0,C 180,E1 16376.686,E2 16376.686} C_VEL
LIN {X 0,Y 345.916,Z 459.708,A -85,B 0,C 180,E1 16372.359,E2 16372.359} C_VEL
LIN {X 0,Y 345.917,Z 459.709,A -85,B 0,C 180,E1 16368.157,E2 16368.157} C_VEL
LIN {X 0,Y 345.922,Z 459.706,A -85,B 0,C 180,E1 16363.89,E2 16363.89} C_VEL
LIN {X 0,Y 345.956,Z 459.979,A -85,B 0,C 180,E1 16360.08,E2 16360.08} C_VEL
LIN {X 0,Y 349.398,Z 468.082,A -85,B 0,C 180,E1 16356.918,E2 16356.918} C_VEL
LIN {X 0,Y 353.543,Z 478.601,A -85,B 0,C 180,E1 16353.339,E2 16353.339} C_VEL
LIN {X 0,Y 357.502,Z 489.855,A -85,B 0,C 180,E1 16349.958,E2 16349.958} C_VEL
LIN {X 0,Y 361.294,Z 502.49,A -85,B 0,C 180,E1 16346.583,E2 16346.583} C_VEL
LIN {X 0,Y 364.489,Z 515.543,A -85,B 0,C 180,E1 16343.468,E2 16343.468} C_VEL
LIN {X 0,Y 360.865,Z 537.831,A -85,B 0,C 180,E1 16339.636,E2 16339.636} C_VEL
LIN {X 0,Y 358.627,Z 553.164,A -85,B 0,C 180,E1 16337.08,E2 16337.08} C_VEL
LIN {X 0,Y 363.888,Z 579.796,A -85,B 0,C 180,E1 16335.767,E2 16335.767} C_VEL
LIN {X 0,Y 365.612,Z 591.428,A -85,B 0,C 180,E1 16335.298,E2 16335.298} C_VEL
LIN {X 0,Y 362.494,Z 683.278,A -85,B 0,C 180,E1 16333.286,E2 16333.286} C_VEL
LIN {X 0,Y 361.644,Z 699.265,A -85,B 0,C 180,E1 16332.649,E2 16332.649} C_VEL
LIN {X 0,Y 360.38,Z 714.475,A -85,B 0,C 180,E1 16331.749,E2 16331.749} C_VEL
LIN {X 0,Y 358.632,Z 729.595,A -85,B 0,C 180,E1 16330.511,E2 16330.511} C_VEL
LIN {X 0,Y 356.729,Z 742.756,A -85,B 0,C 180,E1 16329.097,E2 16329.097} C_VEL
LIN {X 0,Y 354.687,Z 755.103,A -85,B 0,C 180,E1 16327.398,E2 16327.398} C_VEL
LIN {X 0,Y 352.72,Z 765.738,A -85,B 0,C 180,E1 16325.529,E2 16325.529} C_VEL
LIN {X 0,Y 350.796,Z 775.398,A -85,B 0,C 180,E1 16323.37,E2 16323.37} C_VEL
LIN {X 0,Y 349.112,Z 783.338,A -85,B 0,C 180,E1 16321.032,E2 16321.032} C_VEL
LIN {X 0,Y 347.826,Z 789.298,A -85,B 0,C 180,E1 16318.689,E2 16318.689} C_VEL
LIN {X 0,Y 346.836,Z 793.709,A -85,B 0,C 180,E1 16316.172,E2 16316.172} C_VEL
LIN {X 0,Y 346.221,Z 796.375,A -85,B 0,C 180,E1 16313.667,E2 16313.667} C_VEL
LIN {X 0,Y 345.879,Z 797.354,A -85,B 0,C 180,E1 16310.976,E2 16310.976} C_VEL
LIN {X 0,Y 345.821,Z 796.605,A -85,B 0,C 180,E1 16308.369,E2 16308.369} C_VEL
LIN {X 0,Y 346.044,Z 793.825,A -85,B 0,C 180,E1 16305.587,E2 16305.587} C_VEL
LIN {X 0,Y 346.517,Z 789.701,A -85,B 0,C 180,E1 16303.176,E2 16303.176} C_VEL
LIN {X 0,Y 347.362,Z 783.338,A -85,B 0,C 180,E1 16300.615,E2 16300.615} C_VEL
LIN {X 0,Y 348.399,Z 775.953,A -85,B 0,C 180,E1 16298.416,E2 16298.416} C_VEL
LIN {X 0,Y 349.744,Z 766.518,A -85,B 0,C 180,E1 16296.236,E2 16296.236} C_VEL
LIN {X 0,Y 351.195,Z 755.929,A -85,B 0,C 180,E1 16294.327,E2 16294.327} C_VEL
LIN {X 0,Y 352.734,Z 743.884,A -85,B 0,C 180,E1 16292.599,E2 16292.599} C_VEL
LIN {X 0,Y 354.219,Z 730.747,A -85,B 0,C 180,E1 16291.132,E2 16291.132} C_VEL
LIN {X 0,Y 355.554,Z 716.774,A -85,B 0,C 180,E1 16289.919,E2 16289.919} C_VEL
LIN {X 0,Y 356.693,Z 701.007,A -85,B 0,C 180,E1 16288.916,E2 16288.916} C_VEL
LIN {X 0,Y 357.426,Z 685.388,A -85,B 0,C 180,E1 16288.241,E2 16288.241} C_VEL
LIN {X 0,Y 358.043,Z 661.419,A -85,B 0,C 180,E1 16287.654,E2 16287.654} C_VEL
LIN {X 0,Y 359.937,Z 589.687,A -85,B 0,C 180,E1 16286.165,E2 16286.165} C_VEL
LIN {X 0,Y 360.763,Z 589.944,A -85,B 0,C 180,E1 16285.545,E2 16285.545} C_VEL
LIN {X 0,Y 360.763,Z 638.385,A -85,B 0,C 180,E1 16285.545,E2 16285.545} C_VEL
LIN {X 0,Y 355.517,Z 638.385,A -85,B 0,C 180,E1 16283.115,E2 16283.115} C_VEL
LIN {X 0,Y 355.517,Z 556.762,A -85,B 0,C 180,E1 16283.115,E2 16283.115} C_VEL
LIN {X 0,Y 355.517,Z 543.124,A -85,B 0,C 180,E1 16283.115,E2 16283.115} C_VEL
LIN {X 0,Y 355.589,Z 541.695,A -85,B 0,C 180,E1 16283.019,E2 16283.019} C_VEL
LIN {X 0,Y 354.257,Z 545.678,A -85,B 0,C 180,E1 16283.558,E2 16283.558} C_VEL
LIN {X 0,Y 350.581,Z 552.486,A -85,B 0,C 180,E1 16284.15,E2 16284.15} C_VEL
LIN {X 0,Y 348.529,Z 557.947,A -85,B 0,C 180,E1 16284.454,E2 16284.454} C_VEL
LIN {X 0,Y 348.339,Z 562.311,A -85,B 0,C 180,E1 16284.634,E2 16284.634} C_VEL
LIN {X 0,Y 352.701,Z 590.161,A -85,B 0,C 180,E1 16285.62,E2 16285.62} C_VEL
LIN {X 0,Y 350.193,Z 682.85,A -85,B 0,C 180,E1 16287.632,E2 16287.632} C_VEL
LIN {X 0,Y 349.419,Z 699.954,A -85,B 0,C 180,E1 16288.334,E2 16288.334} C_VEL
LIN {X 0,Y 348.34,Z 714.864,A -85,B 0,C 180,E1 16289.26,E2 16289.26} C_VEL
LIN {X 0,Y 346.948,Z 729.578,A -85,B 0,C 180,E1 16290.495,E2 16290.495} C_VEL
LIN {X 0,Y 345.284,Z 743.771,A -85,B 0,C 180,E1 16292.074,E2 16292.074} C_VEL
LIN {X 0,Y 343.706,Z 755.777,A -85,B 0,C 180,E1 16293.79,E2 16293.79} C_VEL
LIN {X 0,Y 342.188,Z 766.401,A -85,B 0,C 180,E1 16295.701,E2 16295.701} C_VEL
LIN {X 0,Y 340.844,Z 775.438,A -85,B 0,C 180,E1 16297.755,E2 16297.755} C_VEL
LIN {X 0,Y 339.626,Z 783.703,A -85,B 0,C 180,E1 16300.174,E2 16300.174} C_VEL
LIN {X 0,Y 338.749,Z 789.891,A -85,B 0,C 180,E1 16302.616,E2 16302.616} C_VEL
LIN {X 0,Y 338.178,Z 794.612,A -85,B 0,C 180,E1 16305.256,E2 16305.256} C_VEL
LIN {X 0,Y 337.916,Z 797.428,A -85,B 0,C 180,E1 16307.922,E2 16307.922} C_VEL
LIN {X 0,Y 337.946,Z 798.548,A -85,B 0,C 180,E1 16310.614,E2 16310.614} C_VEL
LIN {X 0,Y 338.254,Z 797.855,A -85,B 0,C 180,E1 16313.334,E2 16313.334} C_VEL
LIN {X 0,Y 338.862,Z 795.597,A -85,B 0,C 180,E1 16315.893,E2 16315.893} C_VEL
LIN {X 0,Y 339.837,Z 791.532,A -85,B 0,C 180,E1 16318.465,E2 16318.465} C_VEL
LIN {X 0,Y 341.255,Z 785.561,A -85,B 0,C 180,E1 16321.042,E2 16321.042} C_VEL
LIN {X 0,Y 343.062,Z 777.539,A -85,B 0,C 180,E1 16323.534,E2 16323.534} C_VEL
LIN {X 0,Y 344.966,Z 768.735,A -85,B 0,C 180,E1 16325.632,E2 16325.632} C_VEL
LIN {X 0,Y 347.228,Z 757.321,A -85,B 0,C 180,E1 16327.746,E2 16327.746} C_VEL
LIN {X 0,Y 349.323,Z 745.514,A -85,B 0,C 180,E1 16329.451,E2 16329.451} C_VEL
LIN {X 0,Y 351.436,Z 731.999,A -85,B 0,C 180,E1 16330.979,E2 16330.979} C_VEL
LIN {X 0,Y 353.258,Z 717.319,A -85,B 0,C 180,E1 16332.238,E2 16332.238} C_VEL
LIN {X 0,Y 354.678,Z 702.167,A -85,B 0,C 180,E1 16333.2,E2 16333.2} C_VEL
LIN {X 0,Y 355.668,Z 685.339,A -85,B 0,C 180,E1 16333.914,E2 16333.914} C_VEL
LIN {X 0,Y 357.769,Z 626.311,A -85,B 0,C 180,E1 16335.276,E2 16335.276} C_VEL
LIN {X 0,Y 358.869,Z 590.521,A -85,B 0,C 180,E1 16336.064,E2 16336.064} C_VEL
LIN {X 0,Y 353.822,Z 563.172,A -85,B 0,C 180,E1 16337.35,E2 16337.35} C_VEL
LIN {X 0,Y 351.782,Z 552.976,A -85,B 0,C 180,E1 16337.922,E2 16337.922} C_VEL
LIN {X 0,Y 356.012,Z 527.034,A -85,B 0,C 180,E1 16342.372,E2 16342.372} C_VEL
LIN {X 0,Y 357.47,Z 518.742,A -85,B 0,C 180,E1 16343.83,E2 16343.83} C_VEL
LIN {X 0,Y 354.359,Z 505.806,A -85,B 0,C 180,E1 16347.004,E2 16347.004} C_VEL
LIN {X 0,Y 350.824,Z 493.9,A -85,B 0,C 180,E1 16350.27,E2 16350.27} C_VEL
LIN {X 0,Y 347.043,Z 482.866,A -85,B 0,C 180,E1 16353.66,E2 16353.66} C_VEL
LIN {X 0,Y 342.905,Z 472.352,A -85,B 0,C 180,E1 16357.363,E2 16357.363} C_VEL
LIN {X 0,Y 339.474,Z 464.451,A -85,B 0,C 180,E1 16360.56,E2 16360.56} C_VEL
LIN {X 0,Y 337.99,Z 460.788,A -85,B 0,C 180,E1 16362.279,E2 16362.279} C_VEL
LIN {X 0,Y 337.981,Z 460.676,A -85,B 0,C 180,E1 16366.658,E2 16366.658} C_VEL
LIN {X 0,Y 337.984,Z 460.674,A -85,B 0,C 180,E1 16370.979,E2 16370.979} C_VEL
LIN {X 0,Y 337.985,Z 460.672,A -85,B 0,C 180,E1 16375.248,E2 16375.248} C_VEL
LIN {X 0,Y 337.989,Z 460.669,A -85,B 0,C 180,E1 16379.491,E2 16379.491} C_VEL
LIN {X 0,Y 337.985,Z 460.673,A -85,B 0,C 180,E1 16383.731,E2 16383.731} C_VEL
LIN {X 0,Y 337.991,Z 460.685,A -85,B 0,C 180,E1 16387.992,E2 16387.992} C_VEL
LIN {X 0,Y 337.988,Z 460.697,A -85,B 0,C 180,E1 16392.298,E2 16392.298} C_VEL
LIN {X 0,Y 337.986,Z 460.695,A -85,B 0,C 180,E1 16396.569,E2 16396.569} C_VEL
LIN {X 0,Y 337.982,Z 460.689,A -85,B 0,C 180,E1 16400.974,E2 16400.974} C_VEL
LIN {X 0,Y 337.983,Z 460.683,A -85,B 0,C 180,E1 16405.214,E2 16405.214} C_VEL
LIN {X 0,Y 337.991,Z 460.686,A -85,B 0,C 180,E1 16409.605,E2 16409.605} C_VEL
LIN {X 0,Y 338.012,Z 460.888,A -85,B 0,C 180,E1 16413.036,E2 16413.036} C_VEL
LIN {X 0,Y 339.668,Z 464.692,A -85,B 0,C 180,E1 16414.619,E2 16414.619} C_VEL
LIN {X 0,Y 342.636,Z 470.982,A -85,B 0,C 180,E1 16416.951,E2 16416.951} C_VEL
LIN {X 0,Y 346.152,Z 478.448,A -85,B 0,C 180,E1 16419.454,E2 16419.454} C_VEL
LIN {X 0,Y 350.925,Z 489.644,A -85,B 0,C 180,E1 16422.696,E2 16422.696} C_VEL
LIN {X 0,Y 355.792,Z 502.189,A -85,B 0,C 180,E1 16425.818,E2 16425.818} C_VEL
LIN {X 0,Y 360.703,Z 516.672,A -85,B 0,C 180,E1 16428.936,E2 16428.936} C_VEL
LIN {X 0,Y 362.796,Z 523.994,A -85,B 0,C 180,E1 16430.347,E2 16430.347} C_VEL
LIN {X 0,Y 359.17,Z 542.664,A -85,B 0,C 180,E1 16432.637,E2 16432.637} C_VEL
LIN {X 0,Y 362.079,Z 570.662,A -85,B 0,C 180,E1 16433.706,E2 16433.706} C_VEL
LIN {X 0,Y 361.878,Z 583.649,A -85,B 0,C 180,E1 16434.001,E2 16434.001} C_VEL
LIN {X 0,Y 357.307,Z 732.694,A -85,B 0,C 180,E1 16437.037,E2 16437.037} C_VEL
LIN {X 0,Y 355.884,Z 751.094,A -85,B 0,C 180,E1 16437.678,E2 16437.678} C_VEL
LIN {X 0,Y 353.836,Z 769.178,A -85,B 0,C 180,E1 16438.605,E2 16438.605} C_VEL
LIN {X 0,Y 351.519,Z 785.939,A -85,B 0,C 180,E1 16439.771,E2 16439.771} C_VEL
LIN {X 0,Y 348.975,Z 802.184,A -85,B 0,C 180,E1 16441.227,E2 16441.227} C_VEL
LIN {X 0,Y 346.357,Z 817.581,A -85,B 0,C 180,E1 16442.957,E2 16442.957} C_VEL
LIN {X 0,Y 343.777,Z 832.092,A -85,B 0,C 180,E1 16444.965,E2 16444.965} C_VEL
LIN {X 0,Y 341.396,Z 845.863,A -85,B 0,C 180,E1 16447.302,E2 16447.302} C_VEL
LIN {X 0,Y 339.413,Z 858.083,A -85,B 0,C 180,E1 16449.839,E2 16449.839} C_VEL
LIN {X 0,Y 337.935,Z 868.979,A -85,B 0,C 180,E1 16452.613,E2 16452.613} C_VEL
LIN {X 0,Y 337.016,Z 878.326,A -85,B 0,C 180,E1 16455.569,E2 16455.569} C_VEL
LIN {X 0,Y 336.691,Z 885.684,A -85,B 0,C 180,E1 16458.524,E2 16458.524} C_VEL
LIN {X 0,Y 336.77,Z 891.234,A -85,B 0,C 180,E1 16461.463,E2 16461.463} C_VEL
LIN {X 0,Y 337.112,Z 895.091,A -85,B 0,C 180,E1 16464.383,E2 16464.383} C_VEL
LIN {X 0,Y 337.443,Z 897.302,A -85,B 0,C 180,E1 16467.283,E2 16467.283} C_VEL
LIN {X 0,Y 337.595,Z 897.871,A -85,B 0,C 180,E1 16470.17,E2 16470.17} C_VEL
LIN {X 0,Y 337.46,Z 896.776,A -85,B 0,C 180,E1 16473.057,E2 16473.057} C_VEL
LIN {X 0,Y 337.151,Z 893.998,A -85,B 0,C 180,E1 16475.958,E2 16475.958} C_VEL
LIN {X 0,Y 336.854,Z 889.484,A -85,B 0,C 180,E1 16478.879,E2 16478.879} C_VEL
LIN {X 0,Y 336.814,Z 883.145,A -85,B 0,C 180,E1 16481.82,E2 16481.82} C_VEL
LIN {X 0,Y 337.176,Z 874.656,A -85,B 0,C 180,E1 16484.825,E2 16484.825} C_VEL
LIN {X 0,Y 338.019,Z 864.91,A -85,B 0,C 180,E1 16487.561,E2 16487.561} C_VEL
LIN {X 0,Y 339.327,Z 853.492,A -85,B 0,C 180,E1 16490.167,E2 16490.167} C_VEL
LIN {X 0,Y 341.075,Z 840.543,A -85,B 0,C 180,E1 16492.584,E2 16492.584} C_VEL
LIN {X 0,Y 343.046,Z 826.482,A -85,B 0,C 180,E1 16494.725,E2 16494.725} C_VEL
LIN {X 0,Y 345.19,Z 811.514,A -85,B 0,C 180,E1 16496.585,E2 16496.585} C_VEL
LIN {X 0,Y 347.306,Z 795.711,A -85,B 0,C 180,E1 16498.174,E2 16498.174} C_VEL
LIN {X 0,Y 349.447,Z 778.133,A -85,B 0,C 180,E1 16499.562,E2 16499.562} C_VEL
LIN {X 0,Y 351.3,Z 760.2,A -85,B 0,C 180,E1 16500.629,E2 16500.629} C_VEL
LIN {X 0,Y 352.769,Z 741.802,A -85,B 0,C 180,E1 16501.399,E2 16501.399} C_VEL
LIN {X 0,Y 353.537,Z 722.715,A -85,B 0,C 180,E1 16501.896,E2 16501.896} C_VEL
LIN {X 0,Y 357.057,Z 569.943,A -85,B 0,C 180,E1 16504.92,E2 16504.92} C_VEL
LIN {X 0,Y 354.339,Z 542.008,A -85,B 0,C 180,E1 16505.79,E2 16505.79} C_VEL
LIN {X 0,Y 357.925,Z 517.657,A -85,B 0,C 180,E1 16508.668,E2 16508.668} C_VEL
LIN {X 0,Y 351.394,Z 497.21,A -85,B 0,C 180,E1 16512.185,E2 16512.185} C_VEL
LIN {X 0,Y 344.904,Z 478.958,A -85,B 0,C 180,E1 16515.682,E2 16515.682} C_VEL
LIN {X 0,Y 339.12,Z 463.939,A -85,B 0,C 180,E1 16518.891,E2 16518.891} C_VEL
LIN {X 0,Y 338.011,Z 460.805,A -85,B 0,C 180,E1 16519.686,E2 16519.686} C_VEL
LIN {X 0,Y 337.986,Z 460.681,A -85,B 0,C 180,E1 16523.936,E2 16523.936} C_VEL
LIN {X 0,Y 337.981,Z 460.678,A -85,B 0,C 180,E1 16528.225,E2 16528.225} C_VEL
LIN {X 0,Y 337.97,Z 460.676,A -85,B 0,C 180,E1 16532.515,E2 16532.515} C_VEL
LIN {X 0,Y 337.97,Z 460.688,A -85,B 0,C 180,E1 16536.83,E2 16536.83} C_VEL
LIN {X 0,Y 337.972,Z 460.698,A -85,B 0,C 180,E1 16541.208,E2 16541.208} C_VEL
LIN {X 0,Y 337.972,Z 460.667,A -85,B 0,C 180,E1 16545.436,E2 16545.436} C_VEL
LIN {X 0,Y 337.973,Z 460.69,A -85,B 0,C 180,E1 16549.604,E2 16549.604} C_VEL
LIN {X 0,Y 337.986,Z 460.679,A -85,B 0,C 180,E1 16553.887,E2 16553.887} C_VEL
LIN {X 0,Y 337.986,Z 460.674,A -85,B 0,C 180,E1 16558.136,E2 16558.136} C_VEL
LIN {X 0,Y 337.98,Z 460.678,A -85,B 0,C 180,E1 16562.374,E2 16562.374} C_VEL
LIN {X 0,Y 337.975,Z 460.674,A -85,B 0,C 180,E1 16566.626,E2 16566.626} C_VEL
LIN {X 0,Y 337.96,Z 460.677,A -85,B 0,C 180,E1 16570.915,E2 16570.915} C_VEL
LIN {X 0,Y 337.955,Z 460.685,A -85,B 0,C 180,E1 16575.091,E2 16575.091} C_VEL
LIN {X 0,Y 337.944,Z 460.671,A -85,B 0,C 180,E1 16579.352,E2 16579.352} C_VEL
LIN {X 0,Y 337.941,Z 460.692,A -85,B 0,C 180,E1 16583.542,E2 16583.542} C_VEL
LIN {X 0,Y 337.938,Z 460.676,A -85,B 0,C 180,E1 16587.871,E2 16587.871} C_VEL
LIN {X 0,Y 337.936,Z 460.691,A -85,B 0,C 180,E1 16591.98,E2 16591.98} C_VEL
LIN {X 0,Y 337.938,Z 460.69,A -85,B 0,C 180,E1 16596.281,E2 16596.281} C_VEL
LIN {X 0,Y 337.936,Z 460.677,A -85,B 0,C 180,E1 16600.389,E2 16600.389} C_VEL
LIN {X 0,Y 337.939,Z 460.702,A -85,B 0,C 180,E1 16604.525,E2 16604.525} C_VEL
LIN {X 0,Y 337.941,Z 460.682,A -85,B 0,C 180,E1 16608.722,E2 16608.722} C_VEL
LIN {X 0,Y 337.942,Z 460.681,A -85,B 0,C 180,E1 16612.874,E2 16612.874} C_VEL
LIN {X 0,Y 337.949,Z 460.685,A -85,B 0,C 180,E1 16617.167,E2 16617.167} C_VEL
LIN {X 0,Y 337.96,Z 460.685,A -85,B 0,C 180,E1 16621.484,E2 16621.484} C_VEL
LIN {X 0,Y 337.975,Z 460.839,A -85,B 0,C 180,E1 16625.602,E2 16625.602} C_VEL
LIN {X 0,Y 342.263,Z 473.702,A -85,B 0,C 180,E1 16628.941,E2 16628.941} C_VEL
LIN {X 0,Y 346.72,Z 488.227,A -85,B 0,C 180,E1 16632.374,E2 16632.374} C_VEL
LIN {X 0,Y 350.922,Z 503.927,A -85,B 0,C 180,E1 16635.816,E2 16635.816} C_VEL
LIN {X 0,Y 352.439,Z 510.671,A -85,B 0,C 180,E1 16637.215,E2 16637.215} C_VEL
LIN {X 0,Y 348.736,Z 537.834,A -85,B 0,C 180,E1 16641.758,E2 16641.758} C_VEL
